(* IEC 61131-3 sources: Std_PalletMover/Class/MQTTClient_Interface (part 2) *)

      DiagnosticData.LogEvents.Level_Warning  := DiagnosticData.LogEvents.Level_Error;
      DiagnosticData.LogEvents.Level_Info     := DiagnosticData.LogEvents.Level_Error;
      DiagnosticData.LogEvents.Level_Debug    := DiagnosticData.LogEvents.Level_Error;

  end_if;

END_FUNCTION

FUNCTION MQTTClient_Interface::InitMem

END_FUNCTION
//================================================================================================================================================================
//----------------------------------------------------------------END OF INITITALISE METHODS----------------------------------------------------------------------
//================================================================================================================================================================

//================================================================================================================================================================
//-----------------------------------------------------------------SERVER INTERFACE METHODS-----------------------------------------------------------------------
//================================================================================================================================================================
FUNCTION VIRTUAL GLOBAL MQTTClient_Interface::ClientID::Read
	VAR_OUTPUT
		output (EAX) 	: UDINT;
	END_VAR

	ClientID := MQTTClient.ClientID.Read();
	output := ClientID;

END_FUNCTION

FUNCTION VIRTUAL GLOBAL MQTTClient_Interface::ClientID::Write
	VAR_INPUT
		input (EAX) 	: UDINT;
	END_VAR
	VAR_OUTPUT
		result (EAX) 	: UDINT;
	END_VAR

	ClientID := input;
	result := (MQTTClient.ClientID.Write(ClientID))$UDINT;

END_FUNCTION

FUNCTION VIRTUAL GLOBAL MQTTClient_Interface::XMLFilename::Read
	VAR_OUTPUT
		output (EAX) 	: UDINT;
	END_VAR

	XMLFilename := XMLFilenameString.Data.Read();
	output := XMLFilename;

END_FUNCTION

FUNCTION VIRTUAL GLOBAL MQTTClient_Interface::XMLFilename::Write
	VAR_INPUT
		input (EAX) 	: UDINT;
	END_VAR
	VAR_OUTPUT
		result (EAX) 	: UDINT;
	END_VAR

	XMLFilename := input;
	result := (XMLFilenameString.Data.Write(XMLFilename))$UDINT;

END_FUNCTION

FUNCTION VIRTUAL GLOBAL MQTTClient_Interface::ClientActive::Write
	VAR_INPUT
		input (EAX) 	: DINT;
	END_VAR
	VAR_OUTPUT
		result (EAX) 	: DINT;
	END_VAR
  VAR
  	iRetCode : INT;
    tmpPara : DINT;
  END_VAR

  //Falling edge (Disabling Client)
  if (ClientActive = 1) &
     (input = 0)        then

    //If the state is OK
    if InterfaceState = MCIS_Connected         |
       InterfaceState = MCIS_WaitForConnection |
       InterfaceState = MCIS_Reconnecting      then

      //Issue Disconnect Command
      iRetCode := MQTTClient.mqtt_disconnect();

      //Diagnostic Info:
      Diagnostic_Event( Event   :=  DL_LastErrorCode,
                        udValue :=  iRetCode$UDINT);

      if iRetCode <> MQTTClient::MQTT_ERR_SUCCESS$INT then
        Diagnostic_Event( Event   :=  DL_Error,
                          udValue :=  0);
      end_if;

      if iRetCode = MQTTClient::MQTT_ERR_SUCCESS$INT then
        //Create Log: MQTT Client disconnect requested

        Logging_InterfLog(usLevel     :=  MQTTCLIENTINTERFACE_LOGGING_LEVEL_DEBUG,
                          dMsgGroup   :=  MQCLIINF_LOG_DEBUG_CLIENTACTIVE_DISCONNECT_REQUESTED_GRP,
                          dMsgNbr     :=  MQCLIINF_LOG_DEBUG_CLIENTACTIVE_DISCONNECT_REQUESTED_MSG,
                          pMsg        :=  MQCLIINF_LOG_DEBUG_CLIENTACTIVE_DISCONNECT_REQUESTED_TEXT,
                          pPara1      :=  NIL,
                          pPara2      :=  NIL,
                          pPara3      :=  NIL,
                          pPara4      :=  NIL);

      elsif iRetCode = MQTTClient::MQTT_ERR_NO_CONN$INT then
        //Create Log: Requesting MQTT Client Disconnect Failed, no Connection to disconnect.

        Logging_InterfLog(usLevel     :=  MQTTCLIENTINTERFACE_LOGGING_LEVEL_WARNING,
                          dMsgGroup   :=  MQCLIINF_LOG_WARNING_CLIENTACTIVE_DISCONNECT_REQUESTED_GRP,
                          dMsgNbr     :=  MQCLIINF_LOG_WARNING_CLIENTACTIVE_DISCONNECT_REQUESTED_MSG,
                          pMsg        :=  MQCLIINF_LOG_WARNING_CLIENTACTIVE_DISCONNECT_REQUESTED_TEXT,
                          pPara1      :=  NIL,
                          pPara2      :=  NIL,
                          pPara3      :=  NIL,
                          pPara4      :=  NIL);

      else
        //Create Log: Unexpected retcode whilst requesting MQTT Client Disconnect.
        tmpPara := to_dint(iRetCode);

        Logging_InterfLog(usLevel     :=  MQTTCLIENTINTERFACE_LOGGING_LEVEL_ERR,
                          dMsgGroup   :=  MQCLIINF_LOG_WARNING_CLIENTACTIVE_DISCONNECT_UNEXPECTED_RETCODE_GRP,
                          dMsgNbr     :=  MQCLIINF_LOG_WARNING_CLIENTACTIVE_DISCONNECT_UNEXPECTED_RETCODE_MSG,
                          pMsg        :=  MQCLIINF_LOG_WARNING_CLIENTACTIVE_DISCONNECT_UNEXPECTED_RETCODE_TEXT,
                          pPara1      :=  #tmpPara,
                          pPara2      :=  NIL,
                          pPara3      :=  NIL,
                          pPara4      :=  NIL);
      end_if;

    end_if;

    ClientActive := 0;

  else

    ClientActive := input;

  end_if;

	result := ClientActive;

END_FUNCTION
//================================================================================================================================================================
//--------------------------------------------------------------END OF SERVER INTERFACE METHODS-------------------------------------------------------------------
//================================================================================================================================================================

//================================================================================================================================================================
//-----------------------------------------------------------------------CYCLIC METHODS---------------------------------------------------------------------------
//================================================================================================================================================================
FUNCTION VIRTUAL GLOBAL MQTTClient_Interface::CyWork
	VAR_INPUT
		EAX 	: UDINT;
	END_VAR
	VAR_OUTPUT
		state (EAX) 	: UDINT;
	END_VAR

	state := READY;
  MQTTClientInterfaceTask();

END_FUNCTION

FUNCTION MQTTClient_Interface::MQTTClientInterfaceTask
  VAR
  	iRetCode : INT;
    dTemp : DINT;
  END_VAR

  //Set FirstCall if state is changed
  Config.bFirstCall := InterfaceState <> LastState;

  //If not already in Error state, check for errors from interfaces
  if InterfaceState <> MCIS_Error then
    Diagnostic_ReadErrors();
  end_if;

  //=============================================
  //FSM For MQTT Client Interface
  //=============================================
  case InterfaceState of

    //-----------------------------------------------------------------
    //Wait for activation
    //-----------------------------------------------------------------
  	MQTTClient_Interface::t_e_MQTTClientStates::MCIS_Ready:

      if ClientActive = 1 then

        if Config.IsConn.PubTimeout then
          cDataMapPubTimeout := cDataMapPubTimeout.Read();
        end_if;

        if Config.IsConn.SubTimeout then
          cDataMapSubTimeout := cDataMapSubTimeout.Read();
        end_if;

        if Config.IsConn.ConnTimeout then
          cConnectTimeout := cConnectTimeout.Read();
        end_if;

        Logging_InterfLog(usLevel     :=  MQTTCLIENTINTERFACE_LOGGING_LEVEL_INFO,
                          dMsgGroup   :=  MQCLIINF_LOG_INFO_FSM_CLIENT_ACTIVATED_GRP,
                          dMsgNbr     :=  MQCLIINF_LOG_INFO_FSM_CLIENT_ACTIVATED_MSG,
                          pMsg        :=  MQCLIINF_LOG_INFO_FSM_CLIENT_ACTIVATED_TEXT,
                          pPara1      :=  NIL,
                          pPara2      :=  NIL,
                          pPara3      :=  NIL,
                          pPara4      :=  NIL);

        InterfaceState := MCIS_Initialise;

        //Reset Diagnostic Data
        Diagnostic_Event( Event   :=  DL_Reset,
                          udValue :=  0);
      end_if;

      LastState := MCIS_Ready;

    //-----------------------------------------------------------------
    //Initialise, Prepare, Read XML
    //-----------------------------------------------------------------
  	MQTTClient_Interface::t_e_MQTTClientStates::MCIS_Initialise:

      //Perform Init task
      case MCIT_Initialise(bFirstCall:=Config.bFirstCall) of

        TR_Busy:  //Stay in this state

        TR_Done:  //Next State

          InterfaceState := MCIS_Prepare;

        TR_Error: //Go to Error State

          InterfaceState := MCIS_Error;

      end_case;

      LastState := MCIS_Initialise;

    //-----------------------------------------------------------------
    //Prepare Connection, set parameters, initiate Connection
    //-----------------------------------------------------------------
  	MQTTClient_Interface::t_e_MQTTClientStates::MCIS_Prepare:

      //Perform Prepare task
      case MCIT_Prepare(bFirstCall:=Config.bFirstCall) of

        TR_Busy:  //Stay in this state

        TR_Done:  //Create Connection & Next State

          udTimestamp := ops.tAbsolute;

          MQTTClient.mqtt_loop_start();

          iRetCode := MQTTClient.mqtt_connect_async(  host      :=  #MQTTClientConfigData.Config.Connect.aHostname[0],
                                                      port      :=  MQTTClientConfigData.Config.Connect.iPort,
                                                      keepalive :=  MQTTClientConfigData.Config.Connect.iKeepalive);

          //Diagnostic Info:
          Diagnostic_Event( Event   :=  DL_LastErrorCode,
                            udValue :=  iRetCode$UDINT);

          if iRetCode = MQTTClient::MQTT_ERR_SUCCESS$INT then

            InterfaceState := MCIS_WaitForConnection;
            udTimestamp := ops.tAbsolute;

          else

            //Diagnostic Info:
            Diagnostic_Event( Event   :=  DL_Error,
                              udValue :=  0);

            Diagnostic_Event( Event   :=  DL_ConnectFail,
                              udValue :=  0);

            dTemp := to_dint(iRetCode);

            //Create Log Message
            Logging_InterfLog(usLevel     :=  MQTTCLIENTINTERFACE_LOGGING_LEVEL_ERR,
                              dMsgGroup   :=  MQCLIINF_LOG_ERROR_FSM_CONNECTION_FAILED_GRP,
                              dMsgNbr     :=  MQCLIINF_LOG_ERROR_FSM_CONNECTION_FAILED_MSG,
                              pMsg        :=  MQCLIINF_LOG_ERROR_FSM_CONNECTION_FAILED_TEXT,
                              pPara1      :=  #dTemp,
                              pPara2      :=  NIL,
                              pPara3      :=  NIL,
                              pPara4      :=  NIL);

            //Go to Error
            InterfaceState := MCIS_Error;

          end_if;

        TR_Error: //Go to Error State

          InterfaceState := MCIS_Error;

      end_case;

      LastState := MCIS_Prepare;

    //-----------------------------------------------------------------
    //Wait for connection to be made
    //-----------------------------------------------------------------
  	MQTTClient_Interface::t_e_MQTTClientStates::MCIS_WaitForConnection:

      if ops.tAbsolute - udTimestamp >= cConnectTimeout then
        InterfaceState := MCIS_Error;
        //Diagnostic Info:
        Diagnostic_Event( Event   :=  DL_WatchdogTimeout,
                          udValue :=  0);
      end_if;

      LastState := MCIS_WaitForConnection;

    //-----------------------------------------------------------------
    //Wait for connection to be made
    //-----------------------------------------------------------------
  	MQTTClient_Interface::t_e_MQTTClientStates::MCIS_Reconnecting:

      Diagnostic_Calculate();

    //-----------------------------------------------------------------
    //Connected state
    //-----------------------------------------------------------------
  	MQTTClient_Interface::t_e_MQTTClientStates::MCIS_Connected:

      Diagnostic_Calculate();
      DataMap_ProcessMap();

      LastState := MCIS_Connected;

    //-----------------------------------------------------------------
    //Error Occured
    //-----------------------------------------------------------------
  	MQTTClient_Interface::t_e_MQTTClientStates::MCIS_Error:

      //If this is the first cycle in this state
      if LastState <> InterfaceState then
        MQTTClient.mqtt_disconnect();
        udTimestamp := ops.tAbsolute;
      end_if;

      //If Reset
      if (Reset = 1)                                    |
         (cAutoResetTime <> 0                         &
          ops.tAbsolute - udTimestamp >= cAutoResetTime) then
        Reset := 0;
        InterfaceState := MCIS_Ready;
      end_if;

      LastState := MCIS_Error;

  end_case;

END_FUNCTION

FUNCTION MQTTClient_Interface::MCIT_Initialise
  VAR_INPUT
    bFirstCall : BOOL;
  END_VAR
	VAR_OUTPUT
		eRet 	: t_e_TaskRet;
	END_VAR

  //Assume Busy
  eRet := TR_Busy;

  //If first call, restart the FSM
  if bFirstCall then
    States.Initialise := MCSI_Initialize;
  end_if;

  //============================================
  //Initialise FSM
  //============================================
  case States.Initialise of

    //----------------------------------
    //Prepare mem, name and XML Reader
    //----------------------------------
    t_e_MCSInit::MCSI_Initialize:

      //Clear Mem
      SigCLib.MemSet( dst :=  #MQTTClientConfigData,
                      c   :=  0x00,
                      len :=  sizeof(MQTTClientConfigData));

      //If using the XML File, process it
      if Config.IsConn.UseXML then
        cUseXML := cUseXML.Read();
      end_if;

      if cUseXML = 1 then

        //XML Filename
        SigCLib.MemSet( dst :=  #Config.Initialize.aXMLFilename,
                        c   :=  0x00,
                        len :=  sizeof(Config.Initialize.aXMLFilename));
        XMLFilenameString.ReadDataOff(udOff :=  0,
                                      pData :=  #Config.Initialize.aXMLFilename[0],
                                      udMax :=  MQTTCLIENTINTERFACE_MAX_XMLNAME_LEN);
        //Reset Reader
        _XMLReader.Reset();
        _XMLReader.FreeReader();

        States.Initialise := MCSI_ReadXML;

      //If not using the XML File, skip reading & Processing
      else

        States.Initialise := MCSI_AppliConfig;

      end_if;

      //Get Logging Config from Client
      if Config.IsConn.LogConfig then
        cLogConfig := cLogConfig.Read();
      end_if;

    //----------------------------------
    //Read the XML
    //----------------------------------
    t_e_MCSInit::MCSI_ReadXML:

      //Start XML File Read
      if _XMLReader.ReadFile(FileName:=#Config.Initialize.aXMLFilename[0]) then
        States.Initialise := MCSI_WaitForReadXML;
        udTimestamp := ops.tAbsolute;
      else
        //Create Log: Failed to read XML File

        Logging_InterfLog(usLevel     :=  MQTTCLIENTINTERFACE_LOGGING_LEVEL_ERR,
                          dMsgGroup   :=  MQCLIINF_LOG_ERROR_FSM_INIT_READ_FILE_FAILED_GRP,
                          dMsgNbr     :=  MQCLIINF_LOG_ERROR_FSM_INIT_READ_FILE_FAILED_MSG,
                          pMsg        :=  MQCLIINF_LOG_ERROR_FSM_INIT_READ_FILE_FAILED_TEXT,
                          pPara1      :=  NIL,
                          pPara2      :=  NIL,
                          pPara3      :=  NIL,
                          pPara4      :=  NIL);

        States.Initialise := MCSI_Error;
      end_if;

    //----------------------------------
    //Wait for read to finish
    //----------------------------------
    t_e_MCSInit::MCSI_WaitForReadXML:

      //Read Complete
      if _XMLReader.GetXmlState() = _XMLReader::XML_READ_STATE::_STRUCT_CREATED then

        States.Initialise := MCSI_PrepDataMap;

      //Read Error
      elsif _XMLReader.GetXmlState() = _XMLReader::XML_READ_STATE::_ERROR then

        States.Initialise := MCSI_Error;

      //Timeout
      elsif ops.tAbsolute - udTimestamp >= MQTTCLIENTINTERFACE_XML_MAX_READ_TIME then

        States.Initialise := MCSI_Error;

      end_if;

    //----------------------------------
    //Prepare the DataMap - Remove all datamap entries that belong to the XML
    //----------------------------------
    t_e_MCSInit::MCSI_PrepDataMap:

      if Config.pDataMapConfig = NIL then
        //Create Log: Could not initialise, Datamap memory is not OK.

        Logging_InterfLog(usLevel     :=  MQTTCLIENTINTERFACE_LOGGING_LEVEL_ERR,
                          dMsgGroup   :=  MQCLIINF_LOG_ERROR_FSM_INIT_DATAMAP_PTR_GRP,
                          dMsgNbr     :=  MQCLIINF_LOG_ERROR_FSM_INIT_DATAMAP_PTR_MSG,
                          pMsg        :=  MQCLIINF_LOG_ERROR_FSM_INIT_DATAMAP_PTR_TEXT,
                          pPara1      :=  NIL,
                          pPara2      :=  NIL,
                          pPara3      :=  NIL,
                          pPara4      :=  NIL);

        eRet := TR_Error;
        return;
      end_if;

      DataMap_Clear();

      eRet := TR_Busy;
      States.Initialise := MCSI_ProcessXML;

    //----------------------------------
    //Process the XML
    //----------------------------------
    t_e_MCSInit::MCSI_ProcessXML:

      //Process XML
      if ProcessXML() then

        //Update Log Config
        cLogConfig := MQTTClientConfigData.Config.Logging.bdActiveLogs;
        if Config.IsConn.LogConfig then
          cLogConfig.Write(input:=cLogConfig);
        end_if;

        States.Initialise := MCSI_AppliConfig;
        Config.ConfigObject.State := CO_ClientID;

      //Failed
      else

        States.Initialise := MCSI_Error;

      end_if;

    //----------------------------------
    //Call the application config object
    //----------------------------------
    t_e_MCSInit::MCSI_AppliConfig:

      //If an object is logged in
      if Config.ConfigObject.pThis then

        //Process the user config
        case ConfigObject_Process() of
          //------------
          //Keep Calling
          //------------
          TR_Busy:

            eRet := TR_Busy;

          //------------
          //Done, Advance
          //------------
          TR_Done:

            eRet := TR_Done;

          //------------
          //Error Occurred
          //------------
          TR_Error:

            States.Initialise := MCSI_Error;

        end_case;

      else

        eRet := TR_Done;

      end_if;

    //----------------------------------
    //Error Occurred
    //----------------------------------
    t_e_MCSInit::MCSI_Error:

      eRet := TR_Error;

  end_case;

END_FUNCTION

FUNCTION MQTTClient_Interface::MCIT_Prepare
	VAR_INPUT
		bFirstCall 	: BOOL;
	END_VAR
	VAR_OUTPUT
		eRet 	: t_e_TaskRet;
	END_VAR
  VAR
  	iRetCode              : INT;
    pCA, pCert, pKey, pPW : ^CHAR;
    tmpPayLoadSize        : UDINT;
    tmpPara1              : DINT;
    tmpPara2              : DINT;
    tmpPara3              : DINT;
    pID                   : ^UINT;
  END_VAR

  //Assume OK
  eRet := TR_Done;

  //==================================
  //Set the MQTT Class Parameters
  //==================================

    //---------------------------------
    //Client ID
    //---------------------------------
    if MQTTClientConfigData.Config.bClientIDSet then
      pID := #MQTTClientConfigData.Config.aClientID[0];
    else
      pID := NIL;
    end_if;

    iRetCode := MQTTClient.mqtt_reinitialise( id            :=  pID,
                                              clean_session :=  (CleanSession.Read() = 1));

    //Diagnostic Info:
    Diagnostic_Event( Event   :=  DL_LastErrorCode,
                      udValue :=  iRetCode$UDINT);

    if iRetCode <> MQTTClient::MQTT_ERR_SUCCESS$INT then
      Diagnostic_Event( Event   :=  DL_Error,
                        udValue :=  0);
    end_if;
    //- - - - - - - - - - - - - - - - - - - - -
    //Process Reponse
    //- - - - - - - - - - - - - - - - - - - - -
    case iRetCode$MQTTClient::t_e_MQTTErrors of
      //-  -  -  -  -  -  -  -  -  -
      //OK
      //-  -  -  -  -  -  -  -  -  -
      MQTTClient::MQTT_ERR_SUCCESS:

      //-  -  -  -  -  -  -  -  -  -
      //Not OK
      //-  -  -  -  -  -  -  -  -  -
      MQTTClient::MQTT_ERR_NOMEM:

        eRet := TR_Error;
        //Create Log: Error during setting MQTTClient Parameters from XML File, Setting ClientID Failed, Not Enough memory

        Logging_InterfLog(usLevel     :=  MQTTCLIENTINTERFACE_LOGGING_LEVEL_ERR,
                          dMsgGroup   :=  MQCLIINF_LOG_ERROR_FSM_PREP_INIT_FAIL_NOMEM_GRP,
                          dMsgNbr     :=  MQCLIINF_LOG_ERROR_FSM_PREP_INIT_FAIL_NOMEM_MSG,
                          pMsg        :=  MQCLIINF_LOG_ERROR_FSM_PREP_INIT_FAIL_NOMEM_TEXT,
                          pPara1      :=  NIL,
                          pPara2      :=  NIL,
                          pPara3      :=  NIL,
                          pPara4      :=  NIL);
        return;

      //-  -  -  -  -  -  -  -  -  -
      //
      //-  -  -  -  -  -  -  -  -  -
      MQTTClient::MQTT_ERR_INVAL:

        eRet := TR_Error;
        //Create Log: Error during setting MQTTClient Parameters from XML File, Setting ClientID Failed, Input Value / Client State Not OK

        Logging_InterfLog(usLevel     :=  MQTTCLIENTINTERFACE_LOGGING_LEVEL_ERR,
                          dMsgGroup   :=  MQCLIINF_LOG_ERROR_FSM_PREP_INIT_FAIL_INPUT_GRP,
                          dMsgNbr     :=  MQCLIINF_LOG_ERROR_FSM_PREP_INIT_FAIL_INPUT_MSG,
                          pMsg        :=  MQCLIINF_LOG_ERROR_FSM_PREP_INIT_FAIL_INPUT_TEXT,
                          pPara1      :=  NIL,
                          pPara2      :=  NIL,
                          pPara3      :=  NIL,
                          pPara4      :=  NIL);
        return;

    end_case;

    //---------------------------------
    //Connect -> Username & Password
    //---------------------------------
    if MQTTClientConfigData.Config.Connect.ValuesSet.Username then //&
       //MQTTClientConfigData.Config.Connect.ValuesSet.Password then

      iRetCode := MQTTClient.mqtt_username_pw_set(username    :=  #MQTTClientConfigData.Config.Connect.aUsername[0],
                                                  password    :=  #MQTTClientConfigData.Config.Connect.aPassword[0]$BYTE,
                                                  udPassLen   :=  (SigCLib.StrLen16(str0:=#MQTTClientConfigData.Config.Connect.aPassword[0])*sizeof(UINT)));

      //Diagnostic Info:
      Diagnostic_Event( Event   :=  DL_LastErrorCode,
                        udValue :=  iRetCode$UDINT);

      if iRetCode <> MQTTClient::MQTT_ERR_SUCCESS$INT then
        Diagnostic_Event( Event   :=  DL_Error,
                          udValue :=  0);
      end_if;

      //- - - - - - - - - - - - - - - - - - - - -
      //Process Reponse
      //- - - - - - - - - - - - - - - - - - - - -
      case iRetCode$MQTTClient::t_e_MQTTErrors of
        //-  -  -  -  -  -  -  -  -  -
        //OK
        //-  -  -  -  -  -  -  -  -  -
        MQTTClient::MQTT_ERR_SUCCESS:

        //-  -  -  -  -  -  -  -  -  -
        //Not OK
        //-  -  -  -  -  -  -  -  -  -
        MQTTClient::MQTT_ERR_NOMEM:

          eRet := TR_Error;
          //Create Log: Error during setting MQTTClient Parameters from XML File, Setting Username & Password Failed, Not Enough memory

          Logging_InterfLog(usLevel     :=  MQTTCLIENTINTERFACE_LOGGING_LEVEL_ERR,
                            dMsgGroup   :=  MQCLIINF_LOG_ERROR_FSM_PREP_USNPW_FAIL_NOMEM_GRP,
                            dMsgNbr     :=  MQCLIINF_LOG_ERROR_FSM_PREP_USNPW_FAIL_NOMEM_MSG,
                            pMsg        :=  MQCLIINF_LOG_ERROR_FSM_PREP_USNPW_FAIL_NOMEM_TEXT,
                            pPara1      :=  NIL,
                            pPara2      :=  NIL,
                            pPara3      :=  NIL,
                            pPara4      :=  NIL);
          return;

        //-  -  -  -  -  -  -  -  -  -
        //Not OK
        //-  -  -  -  -  -  -  -  -  -
        MQTTClient::MQTT_ERR_INVAL:

          eRet := TR_Error;
          //Create Log: Error during setting MQTTClient Parameters from XML File, Setting Username & Password Failed, Input Value / Client State Not OK

          Logging_InterfLog(usLevel     :=  MQTTCLIENTINTERFACE_LOGGING_LEVEL_ERR,
                            dMsgGroup   :=  MQCLIINF_LOG_ERROR_FSM_PREP_USNPW_FAIL_INPUT_GRP,
                            dMsgNbr     :=  MQCLIINF_LOG_ERROR_FSM_PREP_USNPW_FAIL_INPUT_MSG,
                            pMsg        :=  MQCLIINF_LOG_ERROR_FSM_PREP_USNPW_FAIL_INPUT_TEXT,
                            pPara1      :=  NIL,
                            pPara2      :=  NIL,
                            pPara3      :=  NIL,
                            pPara4      :=  NIL);
          return;

      end_case;

    end_if;

    //---------------------------------
    //Connect -> Max Inflight Messages
    //---------------------------------
    if MQTTClientConfigData.Config.Connect.ValuesSet.MaxInflight then

      iRetCode := MQTTClient.mqtt_max_inflight_messages_set(max_inflight_messages:=MQTTClientConfigData.Config.Connect.iMaxInflightMessages);

      //Diagnostic Info:
      Diagnostic_Event( Event   :=  DL_LastErrorCode,
                        udValue :=  iRetCode$UDINT);

      if iRetCode <> MQTTClient::MQTT_ERR_SUCCESS$INT then
        Diagnostic_Event( Event   :=  DL_Error,
                          udValue :=  0);
      end_if;

      //- - - - - - - - - - - - - - - - - - - - -
      //Process Reponse
      //- - - - - - - - - - - - - - - - - - - - -
      case iRetCode$MQTTClient::t_e_MQTTErrors of
        //-  -  -  -  -  -  -  -  -  -
        //OK
        //-  -  -  -  -  -  -  -  -  -
        MQTTClient::MQTT_ERR_SUCCESS:

        //-  -  -  -  -  -  -  -  -  -
        //Not OK
        //-  -  -  -  -  -  -  -  -  -
        MQTTClient::MQTT_ERR_INVAL:

          eRet := TR_Error;
          //Create Log: Error during setting MQTTClient Parameters from XML File, Setting Max Inflight Messages Failed, Input Value / Client State Not OK
          tmpPara1 := to_dint(MQTTClientConfigData.Config.Connect.iMaxInflightMessages);

          Logging_InterfLog(usLevel     :=  MQTTCLIENTINTERFACE_LOGGING_LEVEL_ERR,
                            dMsgGroup   :=  MQCLIINF_LOG_ERROR_FSM_PREP_SET_INFLIGHT_GRP,
                            dMsgNbr     :=  MQCLIINF_LOG_ERROR_FSM_PREP_SET_INFLIGHT_MSG,
                            pMsg        :=  MQCLIINF_LOG_ERROR_FSM_PREP_SET_INFLIGHT_TEXT,
                            pPara1      :=  #tmpPara1,
                            pPara2      :=  NIL,
                            pPara3      :=  NIL,
                            pPara4      :=  NIL);
          return;

      end_case;

    end_if;

    //---------------------------------
    //Will
    //---------------------------------
    if MQTTClientConfigData.Config.Will.ValuesSet.Topic       &
       MQTTClientConfigData.Config.Will.ValuesSet.Payload     &
       MQTTClientConfigData.Config.Will.ValuesSet.QoS         &
       MQTTClientConfigData.Config.Will.ValuesSet.RetainWill  then

      MQTTClient.mqtt_will_clear();

      tmpPayLoadSize := SigCLib.StrLen(str:=#MQTTClientConfigData.Config.Will.aPayload[0]);

      iRetCode := MQTTClient.mqtt_will_set( topic       :=  #MQTTClientConfigData.Config.Will.aTopic[0],
                                            payloadLen  :=  tmpPayLoadSize,
                                            payload     :=  #MQTTClientConfigData.Config.Will.aPayload[0]$BYTE,
                                            qos         :=  MQTTClientConfigData.Config.Will.iQoS,
                                            retain_will :=  MQTTClientConfigData.Config.Will.bRetain);

      //Diagnostic Info:
      Diagnostic_Event( Event   :=  DL_LastErrorCode,
                        udValue :=  iRetCode$UDINT);

      if iRetCode <> MQTTClient::MQTT_ERR_SUCCESS$INT then
        Diagnostic_Event( Event   :=  DL_Error,
                          udValue :=  0);
      end_if;

      //- - - - - - - - - - - - - - - - - - - - -
      //Process Reponse
      //- - - - - - - - - - - - - - - - - - - - -
      case iRetCode$MQTTClient::t_e_MQTTErrors of
        //-  -  -  -  -  -  -  -  -  -
        //OK
        //-  -  -  -  -  -  -  -  -  -
        MQTTClient::MQTT_ERR_SUCCESS:

        //-  -  -  -  -  -  -  -  -  -
        //Not OK
        //-  -  -  -  -  -  -  -  -  -
        MQTTClient::MQTT_ERR_NOMEM:

          eRet := TR_Error;
          //Create Log: Error during setting MQTTClient Parameters from XML File, Setting Will Failed, Not Enough memory

          Logging_InterfLog(usLevel     :=  MQTTCLIENTINTERFACE_LOGGING_LEVEL_ERR,
                            dMsgGroup   :=  MQCLIINF_LOG_ERROR_FSM_PREP_SET_WILL_NOMEM_GRP,
                            dMsgNbr     :=  MQCLIINF_LOG_ERROR_FSM_PREP_SET_WILL_NOMEM_MSG,
                            pMsg        :=  MQCLIINF_LOG_ERROR_FSM_PREP_SET_WILL_NOMEM_TEXT,
                            pPara1      :=  NIL,
                            pPara2      :=  NIL,
                            pPara3      :=  NIL,
                            pPara4      :=  NIL);
          return;

        //-  -  -  -  -  -  -  -  -  -
        //Not OK
        //-  -  -  -  -  -  -  -  -  -
        MQTTClient::MQTT_ERR_INVAL:

          eRet := TR_Error;
          //Create Log: Error during setting MQTTClient Parameters from XML File, Setting Will Failed, Input Value / Client State Not OK

          Logging_InterfLog(usLevel     :=  MQTTCLIENTINTERFACE_LOGGING_LEVEL_ERR,
                            dMsgGroup   :=  MQCLIINF_LOG_ERROR_FSM_PREP_SET_WILL_INPUT_GRP,
                            dMsgNbr     :=  MQCLIINF_LOG_ERROR_FSM_PREP_SET_WILL_INPUT_MSG,
                            pMsg        :=  MQCLIINF_LOG_ERROR_FSM_PREP_SET_WILL_INPUT_TEXT,
                            pPara1      :=  NIL,
                            pPara2      :=  NIL,
                            pPara3      :=  NIL,
                            pPara4      :=  NIL);
          return;

        //-  -  -  -  -  -  -  -  -  -
        //Not OK
        //-  -  -  -  -  -  -  -  -  -
        MQTTClient::MQTT_ERR_PAYLOAD_SIZE:

          eRet := TR_Error;
          //Create Log: Error during setting MQTTClient Parameters from XML File, Setting Will Failed, Invalid Payload Size

          Logging_InterfLog(usLevel     :=  MQTTCLIENTINTERFACE_LOGGING_LEVEL_ERR,
                            dMsgGroup   :=  MQCLIINF_LOG_ERROR_FSM_PREP_SET_WILL_PAYLOAD_GRP,
                            dMsgNbr     :=  MQCLIINF_LOG_ERROR_FSM_PREP_SET_WILL_PAYLOAD_MSG,
                            pMsg        :=  MQCLIINF_LOG_ERROR_FSM_PREP_SET_WILL_PAYLOAD_TEXT,
                            pPara1      :=  #tmpPayLoadSize$DINT,
                            pPara2      :=  NIL,
                            pPara3      :=  NIL,
                            pPara4      :=  NIL);

          return;

        //-  -  -  -  -  -  -  -  -  -
        //Not OK
        //-  -  -  -  -  -  -  -  -  -
        MQTTClient::MQTT_ERR_MALFORMED_UTF8:

          eRet := TR_Error;
          //Create Log: Error during setting MQTTClient Parameters from XML File, Setting Will Failed, Malformed UTF8

          Logging_InterfLog(usLevel     :=  MQTTCLIENTINTERFACE_LOGGING_LEVEL_ERR,
                            dMsgGroup   :=  MQCLIINF_LOG_ERROR_FSM_PREP_SET_WILL_UTF8_GRP,
                            dMsgNbr     :=  MQCLIINF_LOG_ERROR_FSM_PREP_SET_WILL_UTF8_MSG,
                            pMsg        :=  MQCLIINF_LOG_ERROR_FSM_PREP_SET_WILL_UTF8_TEXT,
                            pPara1      :=  NIL,
                            pPara2      :=  NIL,
                            pPara3      :=  NIL,
                            pPara4      :=  NIL);
          return;

      end_case;

    end_if;

    //---------------------------------
    //Reconnect
    //---------------------------------
    if MQTTClientConfigData.Config.Reconnect.ValuesSet.MinInterval      &
       MQTTClientConfigData.Config.Reconnect.ValuesSet.MaxInterval      &
       MQTTClientConfigData.Config.Reconnect.ValuesSet.ExponentialScale then

      iRetCode := MQTTClient.mqtt_reconnect_delay_set(reconnect_delay             :=  to_uint(MQTTClientConfigData.Config.Reconnect.iMinInterval),
                                                      reconnect_delay_max         :=  to_uint(MQTTClientConfigData.Config.Reconnect.iMaxInterval),
                                                      reconnect_exponential_delay :=  MQTTClientConfigData.Config.Reconnect.bExponential);
      //Diagnostic Info:
      Diagnostic_Event( Event   :=  DL_LastErrorCode,
                        udValue :=  iRetCode$UDINT);

      if iRetCode <> MQTTClient::MQTT_ERR_SUCCESS$INT then
        Diagnostic_Event( Event   :=  DL_Error,
                          udValue :=  0);
      end_if;

      //- - - - - - - - - - - - - - - - - - - - -
      //Process Reponse
      //- - - - - - - - - - - - - - - - - - - - -
      case iRetCode$MQTTClient::t_e_MQTTErrors of
        //-  -  -  -  -  -  -  -  -  -
        //OK
        //-  -  -  -  -  -  -  -  -  -
        MQTTClient::MQTT_ERR_SUCCESS:

        //-  -  -  -  -  -  -  -  -  -
        //Not OK
        //-  -  -  -  -  -  -  -  -  -
        MQTTClient::MQTT_ERR_INVAL:

          eRet := TR_Error;
          //Create Log: Error during setting MQTTClient Parameters from XML File, Setting Reconnect Parameters Failed, Input Value / Client State Not OK

          tmpPara1 := to_dint(MQTTClientConfigData.Config.Reconnect.iMinInterval);
          tmpPara2 := to_dint(MQTTClientConfigData.Config.Reconnect.iMaxInterval);
          tmpPara3 := to_dint(MQTTClientConfigData.Config.Reconnect.bExponential);

          Logging_InterfLog(usLevel     :=  MQTTCLIENTINTERFACE_LOGGING_LEVEL_ERR,
                            dMsgGroup   :=  MQCLIINF_LOG_ERROR_FSM_PREP_SET_RECONNECT_INPUT_GRP,
                            dMsgNbr     :=  MQCLIINF_LOG_ERROR_FSM_PREP_SET_RECONNECT_INPUT_MSG,
                            pMsg        :=  MQCLIINF_LOG_ERROR_FSM_PREP_SET_RECONNECT_INPUT_TEXT,
                            pPara1      :=  #tmpPara1,
                            pPara2      :=  #tmpPara2,
                            pPara3      :=  #tmpPara3,
                            pPara4      :=  NIL);

          return;

      end_case;

    end_if;

    //---------------------------------
    //TLS
    //---------------------------------

    if MQTTClientConfigData.Config.TLS.ValuesSet.TLS then

      pCA := pCert := pKey := pPW := NIL;

      if MQTTClientConfigData.Config.TLS.ValuesSet.CAFile then
        pCA := #MQTTClientConfigData.Config.TLS.aCAFile[0];
      end_if;
      if MQTTClientConfigData.Config.TLS.ValuesSet.CertFile then
        pCert := #MQTTClientConfigData.Config.TLS.aCertFile[0];
      end_if;
      if MQTTClientConfigData.Config.TLS.ValuesSet.KeyFile then
        pKey := #MQTTClientConfigData.Config.TLS.aKeyFile[0];
      end_if;
      if MQTTClientConfigData.Config.TLS.ValuesSet.Password then
        pPW := #MQTTClientConfigData.Config.TLS.aPassword[0];
      end_if;

      iRetCode := MQTTClient.mqtt_tls_set(cafile    :=  pCA,
                                          certfile  :=  pCert,
                                          keyfile   :=  pKey,
                                          pw        :=  pPW);

      //Diagnostic Info:
      Diagnostic_Event( Event   :=  DL_LastErrorCode,
                        udValue :=  iRetCode$UDINT);

      if iRetCode <> MQTTClient::MQTT_ERR_SUCCESS$INT then
        Diagnostic_Event( Event   :=  DL_Error,
                          udValue :=  0);
      end_if;

      //- - - - - - - - - - - - - - - - - - - - -
      //Process Reponse
      //- - - - - - - - - - - - - - - - - - - - -
      case iRetCode$MQTTClient::t_e_MQTTErrors of
        //-  -  -  -  -  -  -  -  -  -
        //OK
        //-  -  -  -  -  -  -  -  -  -
        MQTTClient::MQTT_ERR_SUCCESS:

        //-  -  -  -  -  -  -  -  -  -
        //Not OK
        //-  -  -  -  -  -  -  -  -  -
        MQTTClient::MQTT_ERR_NOMEM:

          eRet := TR_Error;
          //Create Log: Error during setting MQTTClient Parameters from XML File, Setting TLS Data Failed, Not Enough memory

          Logging_InterfLog(usLevel     :=  MQTTCLIENTINTERFACE_LOGGING_LEVEL_ERR,
                            dMsgGroup   :=  MQCLIINF_LOG_ERROR_FSM_PREP_SET_TLS_NOMEM_GRP,
                            dMsgNbr     :=  MQCLIINF_LOG_ERROR_FSM_PREP_SET_TLS_NOMEM_MSG,
                            pMsg        :=  MQCLIINF_LOG_ERROR_FSM_PREP_SET_TLS_NOMEM_TEXT,
                            pPara1      :=  NIL,
                            pPara2      :=  NIL,
                            pPara3      :=  NIL,
                            pPara4      :=  NIL);
          return;

        //-  -  -  -  -  -  -  -  -  -
        //Not OK
        //-  -  -  -  -  -  -  -  -  -
        MQTTClient::MQTT_ERR_INVAL:

          eRet := TR_Error;
          //Create Log: Error during setting MQTTClient Parameters from XML File, Setting TLS Data Failed, Input Value / Client State Not OK

          Logging_InterfLog(usLevel     :=  MQTTCLIENTINTERFACE_LOGGING_LEVEL_ERR,
                            dMsgGroup   :=  MQCLIINF_LOG_ERROR_FSM_PREP_SET_TLS_INPUT_GRP,
                            dMsgNbr     :=  MQCLIINF_LOG_ERROR_FSM_PREP_SET_TLS_INPUT_MSG,
                            pMsg        :=  MQCLIINF_LOG_ERROR_FSM_PREP_SET_TLS_INPUT_TEXT,
                            pPara1      :=  NIL,
                            pPara2      :=  NIL,
                            pPara3      :=  NIL,
                            pPara4      :=  NIL);
          return;

      end_case;

    end_if;

    //===================
    //Set Callbacks
    //===================
    MQTTClient.mqtt_connect_with_flags_callback_set(  pThis                 :=  this,
                                                      on_connect_with_flags :=  #Callback_OnConnectWithFlags());
    MQTTClient.mqtt_disconnect_callback_set(          pThis                 :=  this,
                                                      on_disconnect         :=  #Callback_OnDisconnect());
    MQTTClient.mqtt_publish_callback_set(             pThis                 :=  this,
                                                      on_publish            :=  #Callback_OnPublish());
    MQTTClient.mqtt_message_callback_set(             pThis                 :=  this,
                                                      on_message            :=  #Callback_OnMessage());
    MQTTClient.mqtt_subscribe_callback_set(           pThis                 :=  this,
                                                      on_subscribe          :=  #Callback_OnSubscribe());
    MQTTClient.mqtt_unsubscribe_callback_set(         pThis                 :=  this,
                                                      on_unsubscribe        :=  #Callback_OnUnsubscribe());
    MQTTClient.mqtt_log_callback_set(                 pThis                 :=  this,
                                                      on_log                :=  #Callback_OnLog());
    MQTTClient.mqtt_log_with_detail_callback_set(     pThis                 :=  this,
                                                      on_log_with_detail    :=  #Callback_OnLog_WithDetail());

    //===================
    //Set Logging Filter
    //===================
    if MQTTClientConfigData.Config.Logging.bLogSet then
      _ComLogging.FileLogLevel.Write(input:=MQTTClientConfigData.Config.Logging.bdActiveLogs$UDINT);
      _ComLogging.EventLogLevel.Write(input:=MQTTClientConfigData.Config.Logging.bdActiveLogs$UDINT);
    end_if;

END_FUNCTION
//================================================================================================================================================================
//-------------------------------------------------------------------END OF CYCLIC METHODS------------------------------------------------------------------------
//================================================================================================================================================================

//================================================================================================================================================================
//---------------------------------------------------------------------INTERFACE METHODS--------------------------------------------------------------------------
//================================================================================================================================================================
FUNCTION GLOBAL MQTTClient_Interface::MQTT_Subscribe
	VAR_INPUT
		pTopic 	: ^UINT;
		iQoS 	: INT;
		pThis 	: ^void;
		pCallback 	: ^void;
		pMid 	: ^INT;
		pApplMsgID 	: ^UDINT;
	END_VAR
	VAR_OUTPUT
		retCode 	: INT;
	END_VAR
  VAR
  	iThisMID : INT;
    udThisApplID : UDINT;
    tmpPara, tmpPara2 : DINT;
    pEntry : ^t_s_PubSubEntry;
  END_VAR

  //Assume Error
  retCode := MQTT_ERR_INVAL;

  CriticalSection.SectionStart();

  //Diagnostic Info
  Diagnostic_Event( Event   :=  DL_SubRequest,
                    udValue :=  0);

  //If the input values are not OK
  if pTopic = NIL               |
     iQoS < MQTT_PROT_QOS_MIN   |
     iQoS > MQTT_PROT_QOS_MAX   |
     pThis = NIL                |
     pMid = NIL                 then
    //Create Log: Could not Issue Subscirbe Request, invalid input values.

    tmpPara := to_dint(iQoS);

    Logging_InterfLog(usLevel     :=  MQTTCLIENTINTERFACE_LOGGING_LEVEL_ERR,
                      dMsgGroup   :=  MQCLIINF_LOG_ERROR_SUBSCRIBE_SUB_FAILED_INVALID_INPUT_GRP,
                      dMsgNbr     :=  MQCLIINF_LOG_ERROR_SUBSCRIBE_SUB_FAILED_INVALID_INPUT_MSG,
                      pMsg        :=  MQCLIINF_LOG_ERROR_SUBSCRIBE_SUB_FAILED_INVALID_INPUT_TEXT,
                      pPara1      :=  #pTopic$DINT,
                      pPara2      :=  #tmpPara,
                      pPara3      :=  #pThis$DINT,
                      pPara4      :=  #pCallback$DINT);

    Diagnostic_Event( Event   :=  DL_SubFail,
                      udValue :=  0);

    CriticalSection.SectionStop();
    return;

  end_if;

  //If the interface is not in the correct state
  if InterfaceState < MCIS_Reconnecting |
     InterfaceState > MCIS_Connected    |
     Config.pPubSubConfig = NIL         then

    //Create Log: Could not issue Subscribe Request, The MQTT Interface is not initialized.

    Logging_InterfLog(usLevel     :=  MQTTCLIENTINTERFACE_LOGGING_LEVEL_ERR,
                      dMsgGroup   :=  MQCLIINF_LOG_ERROR_SUBSCRIBE_SUB_FAILED_INTERFACE_STATE_GRP,
                      dMsgNbr     :=  MQCLIINF_LOG_ERROR_SUBSCRIBE_SUB_FAILED_INTERFACE_STATE_MSG,
                      pMsg        :=  MQCLIINF_LOG_ERROR_SUBSCRIBE_SUB_FAILED_INTERFACE_STATE_TEXT,
                      pPara1      :=  #InterfaceState$DINT,
                      pPara2      :=  NIL,
                      pPara3      :=  NIL,
                      pPara4      :=  NIL);

    Diagnostic_Event( Event   :=  DL_SubFail,
                      udValue :=  0);

    CriticalSection.SectionStop();
    return;

  end_if;

  //If there is no more space in the list
  if Config.pPubSubConfig^.PubSubList.udNumEntries >= Config.pPubSubConfig^.PubSubList.udMaxEntries - 1 then

    retCode := MQTT_ERR_NOMEM;
    //Create Log: Could not issue subscribe request, MQTT Interface PubSubList is Full.

    tmpPara   := to_dint(Config.pPubSubConfig^.PubSubList.udMaxEntries);
    tmpPara2  := to_dint(Config.pPubSubConfig^.PubSubList.udNumEntries);

    Logging_InterfLog(usLevel     :=  MQTTCLIENTINTERFACE_LOGGING_LEVEL_ERR,
                      dMsgGroup   :=  MQCLIINF_LOG_ERROR_SUBSCRIBE_SUB_FAILED_LIST_FULL_GRP,
                      dMsgNbr     :=  MQCLIINF_LOG_ERROR_SUBSCRIBE_SUB_FAILED_LIST_FULL_MSG,
                      pMsg        :=  MQCLIINF_LOG_ERROR_SUBSCRIBE_SUB_FAILED_LIST_FULL_TEXT,
                      pPara1      :=  #tmpPara2,
                      pPara2      :=  #tmpPara,
                      pPara3      :=  NIL,
                      pPara4      :=  NIL);

    Diagnostic_Event( Event   :=  DL_SubFail,
                      udValue :=  0);

    CriticalSection.SectionStop();
    return;

  end_if;

  //========================
  //Add the QoS Diag Event
  //========================
  case iQos of
    //---------
    //QoS 0
    //---------
    0:
        Diagnostic_Event( Event   :=  DL_Sub0,
                          udValue :=  0);

    //---------
    //QoS 1
    //---------
    1:
        Diagnostic_Event( Event   :=  DL_Sub1,
                          udValue :=  0);

    //---------
    //QoS 2
    //---------
    2:
        Diagnostic_Event( Event   :=  DL_Sub2,
                          udValue :=  0);
  end_case;

  // Check if the subscription already exists, if so just return Already Subscribed
  udThisApplID := PubSub_CheckSubscription( pTopic    :=  pTopic,
                                            pThis     :=  pThis,
                                            pCallback :=  pCallback);

  if udThisApplID > 0 then

    tmpPara := to_dint(udThisApplID);

    Logging_InterfLog(usLevel     :=  MQTTCLIENTINTERFACE_LOGGING_LEVEL_INFO,
                      dMsgGroup   :=  MQCLIINF_LOG_INFO_SUBSCRIBE_ALREADY_SUBSCRIBED_GRP,
                      dMsgNbr     :=  MQCLIINF_LOG_INFO_SUBSCRIBE_ALREADY_SUBSCRIBED_MSG,
                      pMsg        :=  MQCLIINF_LOG_INFO_SUBSCRIBE_ALREADY_SUBSCRIBED_TEXT,
                      pPara1      :=  #tmpPara,
                      pPara2      :=  NIL,
                      pPara3      :=  NIL,
                      pPara4      :=  NIL);

    retCode := MQTTClient::MQTT_ERR_ALREADY_SUB;

    CriticalSection.SectionStop();
    return;

  end_if;

  iThisMID      := Counters_GetSubMID();
  udThisApplID  := Counters_GetApplID();

  //Subscribe
  retCode := MQTTClient.mqtt_subscribe(mid        :=  #iThisMID,
                                       subscribe  :=  pTopic,
                                       qos        :=  iQoS);

  //Diagnostic Info:
  Diagnostic_Event( Event   :=  DL_LastErrorCode,
                    udValue :=  retCode$UDINT);

  //If the MQTT Client accepts the subscription, log the subscription to the PubSub List
  if retCode = MQTT_ERR_SUCCESS$INT then

    pEntry := (Config.pPubSubConfig^.PubSubList.pEntries$UDINT + sizeof(t_s_PubSubEntry)*Config.pPubSubConfig^.PubSubList.udNumEntries)$^t_s_PubSubEntry;

    pEntry^.iMid             := iThisMID;
    pEntry^.EntryType        := PSE_Subscribe;
    pEntry^.Callback.pThis   := pThis;
    pEntry^.Callback.pMethod := pCallback;
    pEntry^.udAppliID        := udThisApplID;
    pEntry^.iUnsubMid        := -1;

    if pApplMsgID then
      pApplMsgID^ := udThisApplID;
    end_if;

    if pMid then
      pMid^ := iThisMID;
    end_if;

    SigCLib.MemSet( dst :=  #pEntry^.aTopic[0],
                    c   :=  0x00,
                    len :=  sizeof(t_s_PubSubEntry.aTopic));
    SigCLib.StrCpy16( dst0  :=  #pEntry^.aTopic[0],
                      src0  :=  pTopic);

    Config.pPubSubConfig^.PubSubList.udNumEntries += 1;
    Counters_IncSubMID();
    Counters_IncApplID();

    //Create Log: Successfully issued Subscribe Request.

    tmpPara := to_dint(iThisMID);

    Logging_InterfLog(usLevel     :=  MQTTCLIENTINTERFACE_LOGGING_LEVEL_INFO,
                      dMsgGroup   :=  MQCLIINF_LOG_INFO_SUBSCRIBE_ENTRY_ADDED_GRP,
                      dMsgNbr     :=  MQCLIINF_LOG_INFO_SUBSCRIBE_ENTRY_ADDED_MSG,
                      pMsg        :=  MQCLIINF_LOG_INFO_SUBSCRIBE_ENTRY_ADDED_TEXT,
                      pPara1      :=  #tmpPara,
                      pPara2      :=  NIL,
                      pPara3      :=  NIL,
                      pPara4      :=  NIL);

  else

    Logging_InterfLog(usLevel     :=  MQTTCLIENTINTERFACE_LOGGING_LEVEL_ERR,
                      dMsgGroup   :=  MQCLIINF_LOG_ERROR_SUBSCRIBE_SUB_FAILED_GRP,
                      dMsgNbr     :=  MQCLIINF_LOG_ERROR_SUBSCRIBE_SUB_FAILED_MSG,
                      pMsg        :=  MQCLIINF_LOG_ERROR_SUBSCRIBE_SUB_FAILED_TEXT,
                      pPara1      :=  #tmpPara,
                      pPara2      :=  NIL,
                      pPara3      :=  NIL,
                      pPara4      :=  NIL);

    //Diagnostic Data
    Diagnostic_Event( Event   :=  DL_Error,
                      udValue :=  0);
    Diagnostic_Event( Event   :=  DL_SubFail,
                      udValue :=  0);

  end_if;

  CriticalSection.SectionStop();

END_FUNCTION

FUNCTION GLOBAL MQTTClient_Interface::MQTT_Publish
	VAR_INPUT
		pTopic 	: ^UINT;
		iQoS 	: INT;
		pPayload 	: ^void;
		udPayloadLen 	: UDINT;
		bRetain 	: BOOL;
		pThis 	: ^void;
		pCallback 	: ^void;
		pMid 	: ^INT;
		pApplMsgID 	: ^UDINT;
	END_VAR
	VAR_OUTPUT
		retCode 	: INT;
	END_VAR
  VAR
    iRetCode : INT;
  	iThisMID : INT;
    udThisApplID : UDINT;
    tmpPara, tmpPara2 : DINT;
    pEntry : ^t_s_PubSubEntry;
  END_VAR

  CriticalSection.SectionStart();

  //Assume Fail
  retCode := MQTT_ERR_INVAL;

  Diagnostic_Event( Event   :=  DL_PubRequest,
                    udValue :=  0);

  //Check input values
  if pTopic = NIL                                                                 |
     SigCLib.StrLen16(str0:=pTopic) > MQTTCLIENTINTERFACE_PUBSUB_TOPIC_MAX_LEN    |
     iQoS > MQTT_PROT_QOS_MAX                                                     |
     iQos < MQTT_PROT_QOS_MIN                                                     |
     udPayloadLen > MQTTCLIENT_MAX_DATA_LEN                                       |
     ((pPayload <> NIL) & (udPayloadLen = 0))                                     then
    //Create Log: Failed to issue publish request, invalid input values.

    tmpPara := to_dint(iQoS);

    Logging_InterfLog(usLevel     :=  MQTTCLIENTINTERFACE_LOGGING_LEVEL_ERR,
                      dMsgGroup   :=  MQCLIINF_LOG_ERROR_PUBLISH_PUB_FAILED_INVALID_INPUT_GRP,
                      dMsgNbr     :=  MQCLIINF_LOG_ERROR_PUBLISH_PUB_FAILED_INVALID_INPUT_MSG,
                      pMsg        :=  MQCLIINF_LOG_ERROR_PUBLISH_PUB_FAILED_INVALID_INPUT_TEXT,
                      pPara1      :=  #pTopic$DINT,
                      pPara2      :=  #tmpPara,
                      pPara3      :=  #udPayloadLen$DINT,
                      pPara4      :=  #pPayload$DINT);

    Diagnostic_Event( Event   :=  DL_PubFail,
                      udValue :=  0);

    return;

  end_if;

  //Check the state
  if InterfaceState < MCIS_Reconnecting |
     InterfaceState > MCIS_Connected    |
     Config.pPubSubConfig = NIL         then

    retCode := MQTT_ERR_NO_CONN;

    //Create Log: Failed to issue publish request, no Connection MQTT Broker or the MQTT interface class is not initialised.

    Logging_InterfLog(usLevel     :=  MQTTCLIENTINTERFACE_LOGGING_LEVEL_ERR,
                      dMsgGroup   :=  MQCLIINF_LOG_ERROR_PUBLISH_PUB_FAILED_INTERFACE_STATE_GRP,
                      dMsgNbr     :=  MQCLIINF_LOG_ERROR_PUBLISH_PUB_FAILED_INTERFACE_STATE_MSG,
                      pMsg        :=  MQCLIINF_LOG_ERROR_PUBLISH_PUB_FAILED_INTERFACE_STATE_TEXT,
                      pPara1      :=  #InterfaceState$DINT,
                      pPara2      :=  NIL,
                      pPara3      :=  NIL,
                      pPara4      :=  NIL);

    Diagnostic_Event( Event   :=  DL_PubFail,
                      udValue :=  0);

    return;

  end_if;

  //If there is no more space in the list
  if Config.pPubSubConfig^.PubSubList.udNumEntries >= Config.pPubSubConfig^.PubSubList.udMaxEntries - 1 then

    retCode := MQTT_ERR_NOMEM;

    Diagnostic_Event( Event   :=  DL_PubFail,
                      udValue :=  0);

    tmpPara   := to_dint(Config.pPubSubConfig^.PubSubList.udMaxEntries);
    tmpPara2  := to_dint(Config.pPubSubConfig^.PubSubList.udNumEntries);

    Logging_InterfLog(usLevel     :=  MQTTCLIENTINTERFACE_LOGGING_LEVEL_ERR,
                      dMsgGroup   :=  MQCLIINF_LOG_ERROR_SUBSCRIBE_SUB_FAILED_LIST_FULL_GRP,
                      dMsgNbr     :=  MQCLIINF_LOG_ERROR_SUBSCRIBE_SUB_FAILED_LIST_FULL_MSG,
                      pMsg        :=  MQCLIINF_LOG_ERROR_SUBSCRIBE_SUB_FAILED_LIST_FULL_TEXT,
                      pPara1      :=  #tmpPara2,
                      pPara2      :=  #tmpPara,
                      pPara3      :=  NIL,
                      pPara4      :=  NIL);

    return;

  end_if;

  udThisApplID  := Counters_GetApplID();

  iRetCode := MQTTClient.mqtt_publish(mid         :=  #iThisMID,
                                      topic       :=  pTopic,
                                      payloadLen  :=  udPayloadLen,
                                      payload     :=  pPayload,
                                      qos         :=  iQoS,
                                      retain_pub  :=  bRetain);

  //Diagnostic Info:
  Diagnostic_Event( Event   :=  DL_LastErrorCode,
                    udValue :=  retCode$UDINT);

  if iRetCode <> MQTT_ERR_SUCCESS$INT then

    retCode := iRetCode;

    tmpPara := to_dint(retCode);

    Logging_InterfLog(usLevel     :=  MQTTCLIENTINTERFACE_LOGGING_LEVEL_ERR,
                      dMsgGroup   :=  MQCLIINF_LOG_ERROR_SUBSCRIBE_SUB_FAILED_GRP,
                      dMsgNbr     :=  MQCLIINF_LOG_ERROR_SUBSCRIBE_SUB_FAILED_MSG,
                      pMsg        :=  MQCLIINF_LOG_ERROR_SUBSCRIBE_SUB_FAILED_TEXT,
                      pPara1      :=  #tmpPara,
                      pPara2      :=  NIL,
                      pPara3      :=  NIL,
                      pPara4      :=  NIL);

    Diagnostic_Event( Event   :=  DL_PubFail,
                      udValue :=  0);

    Diagnostic_Event( Event   :=  DL_Error,
                      udValue :=  0);

    return;

  end_if;

  Counters_IncPubMID();
  Counters_IncApplID();

  //========================
  //Add the QoS Diag Event
  //========================
  case iQos of
    //---------
    //QoS 0
    //---------
    0:
        Diagnostic_Event( Event   :=  DL_Pub0,
                          udValue :=  0);

    //---------
    //QoS 1
    //---------
    1:
        Diagnostic_Event( Event   :=  DL_Pub1,
                          udValue :=  0);

    //---------
    //QoS 2
    //---------
    2:
        Diagnostic_Event( Event   :=  DL_Pub2,
                          udValue :=  0);
  end_case;

  Diagnostic_Event( Event   :=  DL_TXBytes,
                    udValue :=  udPayloadLen);

  //Add to the PubSubList

  pEntry := (Config.pPubSubConfig^.PubSubList.pEntries$UDINT + sizeof(t_s_PubSubEntry)*Config.pPubSubConfig^.PubSubList.udNumEntries)$^t_s_PubSubEntry;

  pEntry^.iMid             := iThisMID;
  pEntry^.EntryType        := PSE_Publish;
  pEntry^.udAppliID        := udThisApplID;
  pEntry^.Callback.pThis   := pThis;
  pEntry^.Callback.pMethod := pCallback;
  pEntry^.iUnsubMid        := -1;

  SigCLib.MemSet( dst :=  #pEntry^.aTopic,
                  c   :=  0x00,
                  len :=  sizeof(t_s_PubSubEntry.aTopic));

  SigCLib.StrCpy16( dst0  :=  #pEntry^.aTopic[0],
                    src0  :=  pTopic);

  if pMid then
    pMid^ := iThisMID;
  end_if;
  if pApplMsgID then
    pApplMsgID^:= udThisApplID;
  end_if;

  Config.pPubSubConfig^.PubSubList.udNumEntries += 1;

  retCode := MQTT_ERR_SUCCESS;

  CriticalSection.SectionStop();

END_FUNCTION

FUNCTION GLOBAL MQTTClient_Interface::MQTT_Unsubscribe
	VAR_INPUT
		pApplMsgID 	: ^UDINT;
		pTopic 	: ^UINT;
		pMid 	: ^INT;
		pThis 	: ^void;
		pCallback 	: ^void;
	END_VAR
	VAR_OUTPUT
		retCode 	: INT;
	END_VAR
  VAR
    iThisMID : INT;
  	udApplMsgID, udCount, udCount2 : UDINT;
    pPubSubEntry, pPubSubSearchEntry : ^t_s_PubSubEntry;
    bTopicFound, bSubscriptionFound : BOOL;
    tmpPara : DINT;
  END_VAR

  //Assume Error
  retCode := MQTT_ERR_INVAL;

  Diagnostic_Event( Event   :=  DL_UnsubRequest,
                    udValue :=  0);

  //If the input is oK
  if (pApplMsgID | pTopic)                                &
     Config.pPubSubConfig                                 &
     (Config.pPubSubConfig^.PubSubList.udNumEntries > 0)  then

    udApplMsgID := 0;
    bTopicFound := TRUE;

    //1. Determine the Application Message ID:

    //==========================================================
    //Based on the input, determine the ApplMsgID to Unsubscribe
    //==========================================================
      //-----------------------------------
      //Both are set, Use the ApplMsgID
      //-----------------------------------
      if pApplMsgID &
         pTopic then

        udApplMsgID := pApplMsgID^;

      //-----------------------------------
      //Only ApplMsgID is set, use this
      //-----------------------------------
      elsif pApplMsgID      &
            (pTopic = NIL)  then

        udApplMsgID := pApplMsgID^;

      //-----------------------------------
      //Only Topic is set, Determine ApplMsgID
      //-----------------------------------
      elsif pTopic              &
            (pApplMsgID = NIL)  then

        pPubSubEntry := Config.pPubSubConfig^.PubSubList.pEntries;

        for udCount := 0 to Config.pPubSubConfig^.PubSubList.udNumEntries - 1 do

          if SigCLib.StrCmp16(src1:=pTopic, src2:=#pPubSubEntry^.aTopic[0]) = 0 then
            udApplMsgID := pPubSubEntry^.udAppliID;
            bTopicFound := TRUE;
            exit;
          end_if;

          pPubSubEntry$UDINT += sizeof(t_s_PubSubEntry);

        end_for;

        if bTopicFound = FALSE then
          //Create Log: Failed to perform Unsubscribe command, Could not find the Subscription in the PubSubList.

          Logging_InterfLog(usLevel     :=  MQTTCLIENTINTERFACE_LOGGING_LEVEL_ERR,
                            dMsgGroup   :=  MQCLIINF_LOG_ERROR_UNSUBSCRIBE_UNSUB_FAILED_NOT_FOUND_GRP,
                            dMsgNbr     :=  MQCLIINF_LOG_ERROR_UNSUBSCRIBE_UNSUB_FAILED_NOT_FOUND_MSG,
                            pMsg        :=  MQCLIINF_LOG_ERROR_UNSUBSCRIBE_UNSUB_FAILED_NOT_FOUND_TEXT,
                            pPara1      :=  NIL,
                            pPara2      :=  NIL,
                            pPara3      :=  NIL,
                            pPara4      :=  NIL);

          Diagnostic_Event( Event   :=  DL_UnsubFail,
                            udValue :=  0);

          return;
        end_if;

      end_if;

    //2. Find and Unsubscribe the Message

    pPubSubEntry := Config.pPubSubConfig^.PubSubList.pEntries;

    for udCount := 0 to Config.pPubSubConfig^.PubSubList.udNumEntries - 1 do

      if pPubSubEntry^.udAppliID = udApplMsgID then

        //See if this topic is still subscribed to by any other parties, if so, do not unsubscribe
        bSubscriptionFound := FALSE;

        pPubSubSearchEntry$UDINT := (Config.pPubSubConfig^.PubSubList.pEntries)$UDINT;

        for udCount2 := 0 to Config.pPubSubConfig^.PubSubList.udNumEntries - 1 do

          if (udCount2 <> udCount) &
             SigCLib.StrCmp16(src1:=#pPubSubEntry^.aTopic[0], src2:=#pPubSubSearchEntry^.aTopic[0]) = 0 then

            //Create Log: Unsubscribe: Unsubscribe requested for a topic where atleast one other party in the application is still subscribed, the Unsubscribe request will not be sent
            Logging_InterfLog(usLevel     :=  MQTTCLIENTINTERFACE_LOGGING_LEVEL_DEBUG,
                              dMsgGroup   :=  MQCLIINF_LOG_DEBUG_UNSUBSCRIBE_STILL_SUBSCRIBED_GRP,
                              dMsgNbr     :=  MQCLIINF_LOG_DEBUG_UNSUBSCRIBE_STILL_SUBSCRIBED_MSG,
                              pMsg        :=  MQCLIINF_LOG_DEBUG_UNSUBSCRIBE_STILL_SUBSCRIBED_TEXT,
                              pPara1      :=  #pPubSubEntry^.udAppliID$DINT,
                              pPara2      :=  #pPubSubSearchEntry^.udAppliID$DINT,
                              pPara3      :=  NIL,
                              pPara4      :=  NIL);

            bSubscriptionFound := TRUE;
            exit;

          end_if;

          pPubSubSearchEntry$UDINT += sizeof(t_s_PubSubEntry);

        end_for;

        iThisMID := Counters_GetSubMID();

        pPubSubEntry^.iUnsubMid := iThisMID;

        if pMid then
          pMid^ := iThisMID;
        end_if;

        Counters_IncSubMID();

        //If no other subscription was found for this topic, unsubscribe
        if bSubscriptionFound = FALSE then

          retCode := MQTTClient.mqtt_unsubscribe( mid   :=  #pPubSubEntry^.iUnsubMid,
                                                  unsub :=  #pPubSubEntry^.aTopic[0]);

          //Diagnostic Info:
          Diagnostic_Event( Event   :=  DL_LastErrorCode,
                            udValue :=  retCode$UDINT);

          if retCode <> MQTTClient::MQTT_ERR_SUCCESS$INT then

            Diagnostic_Event( Event   :=  DL_UnsubFail,
                              udValue :=  0);
            Diagnostic_Event( Event   :=  DL_Error,
                              udValue :=  0);

          end_if;

          //====================
          //Act on RetCode
          //====================
          case retCode$MQTTClient::t_e_MQTTErrors of
            //-----------------
            //OK
            //-----------------
            MQTT_ERR_SUCCESS:

              //Save Callback Data if set
              if pCallback &
                 pThis     then

                pPubSubEntry^.Callback.pThis    := pThis;
                pPubSubEntry^.Callback.pMethod  := pCallback;

              //Callback data not set but also no pre-existing callback data, the user will receive no feedback
              elsif pPubSubEntry^.Callback.pThis    = NIL |
                    pPubSubEntry^.Callback.pMethod  = NIL then

                //Create Log: No Callback details specified during Unsubscribe, also no pre existing details, no callback possible.

                tmpPara := to_dint(iThisMID);

                Logging_InterfLog(usLevel     :=  MQTTCLIENTINTERFACE_LOGGING_LEVEL_WARNING,
                                  dMsgGroup   :=  MQCLIINF_LOG_WARNING_UNSUBSCRIBE_CALLBACK_NOTSET_GRP,
                                  dMsgNbr     :=  MQCLIINF_LOG_WARNING_UNSUBSCRIBE_CALLBACK_NOTSET_MSG,
                                  pMsg        :=  MQCLIINF_LOG_WARNING_UNSUBSCRIBE_CALLBACK_NOTSET_TEXT,
                                  pPara1      :=  #udApplMsgID$DINT,
                                  pPara2      :=  #tmpPara,
                                  pPara3      :=  NIL,
                                  pPara4      :=  NIL);

              end_if;

              //Create Log: Successfully issued the unsubscribe request for...

              tmpPara := to_dint(iThisMID);

              Logging_InterfLog(usLevel     :=  MQTTCLIENTINTERFACE_LOGGING_LEVEL_INFO,
                                dMsgGroup   :=  MQCLIINF_LOG_INFO_UNSUBSCRIBE_ENTRY_ADDED_GRP,
                                dMsgNbr     :=  MQCLIINF_LOG_INFO_UNSUBSCRIBE_ENTRY_ADDED_MSG,
                                pMsg        :=  MQCLIINF_LOG_INFO_UNSUBSCRIBE_ENTRY_ADDED_TEXT,
                                pPara1      :=  #udApplMsgID$DINT,
                                pPara2      :=  #tmpPara,
                                pPara3      :=  NIL,
                                pPara4      :=  NIL);

            //-----------------
            //Error
            //-----------------
            MQTT_ERR_INVAL:

              //Create Log: Unsubscribe failed, input values not accepted

              tmpPara := to_dint(iThisMID);

              Logging_InterfLog(usLevel     :=  MQTTCLIENTINTERFACE_LOGGING_LEVEL_ERR,
                                dMsgGroup   :=  MQCLIINF_LOG_ERROR_UNSUBSCRIBE_UNSUB_REQ_FAILED_INPUT_GRP,
                                dMsgNbr     :=  MQCLIINF_LOG_ERROR_UNSUBSCRIBE_UNSUB_REQ_FAILED_INPUT_MSG,
                                pMsg        :=  MQCLIINF_LOG_ERROR_UNSUBSCRIBE_UNSUB_REQ_FAILED_INPUT_TEXT,
                                pPara1      :=  #udApplMsgID$DINT,
                                pPara2      :=  #tmpPara,
                                pPara3      :=  NIL,
                                pPara4      :=  NIL);

            //-----------------
            //Retry
            //-----------------
            MQTT_ERR_NO_CONN:

              //Create Log: Unsubscribe failed, no connection mqtt client

              tmpPara := to_dint(iThisMID);

              Logging_InterfLog(usLevel     :=  MQTTCLIENTINTERFACE_LOGGING_LEVEL_ERR,
                                dMsgGroup   :=  MQCLIINF_LOG_ERROR_UNSUBSCRIBE_UNSUB_FAILED_CONN_GRP,
                                dMsgNbr     :=  MQCLIINF_LOG_ERROR_UNSUBSCRIBE_UNSUB_FAILED_CONN_MSG,
                                pMsg        :=  MQCLIINF_LOG_ERROR_UNSUBSCRIBE_UNSUB_FAILED_CONN_TEXT,
                                pPara1      :=  #udApplMsgID$DINT,
                                pPara2      :=  #tmpPara,
                                pPara3      :=  NIL,
                                pPara4      :=  NIL);

            //-----------------
            //Retry
            //-----------------
            MQTT_ERR_NOMEM:

              //Create Log: Unsubscribe failed, no space in message buffer

              tmpPara := to_dint(iThisMID);

              Logging_InterfLog(usLevel     :=  MQTTCLIENTINTERFACE_LOGGING_LEVEL_ERR,
                                dMsgGroup   :=  MQCLIINF_LOG_ERROR_UNSUBSCRIBE_UNSUB_FAILED_NOMEM_GRP,
                                dMsgNbr     :=  MQCLIINF_LOG_ERROR_UNSUBSCRIBE_UNSUB_FAILED_NOMEM_MSG,
                                pMsg        :=  MQCLIINF_LOG_ERROR_UNSUBSCRIBE_UNSUB_FAILED_NOMEM_TEXT,
                                pPara1      :=  #udApplMsgID$DINT,
                                pPara2      :=  #tmpPara,
                                pPara3      :=  NIL,
                                pPara4      :=  NIL);
          //All other
          else

            tmpPara := to_dint(retCode);

            Logging_InterfLog(usLevel     :=  MQTTCLIENTINTERFACE_LOGGING_LEVEL_ERR,
                              dMsgGroup   :=  MQCLIINF_LOG_ERROR_UNSUBSCRIBE_UNSUB_FAILED_GRP,
                              dMsgNbr     :=  MQCLIINF_LOG_ERROR_UNSUBSCRIBE_UNSUB_FAILED_MSG,
                              pMsg        :=  MQCLIINF_LOG_ERROR_UNSUBSCRIBE_UNSUB_FAILED_TEXT,
                              pPara1      :=  #tmpPara,
                              pPara2      :=  NIL,
                              pPara3      :=  NIL,
                              pPara4      :=  NIL);

          end_case;

          return;

        //Someone else is still subscribed to this data.
        else

          //Perform the Unsubscribed callback for this entry if it is set
          //(Even though we did not send an Unsubscribe Request we must let the requesting party know that we handled their request)
          if pPubSubEntry^.Callback.pThis   &
             pPubSubEntry^.Callback.pMethod then

            pPubSubEntry^.Callback.pMethod$PubSub_Callback(pThis        :=  pPubSubEntry^.Callback.pThis,
                                                           MsgType      :=  PSRC_Unsubscribed,
                                                           iMid         :=  pPubSubEntry^.iUnsubMid,
                                                           iGrantedQoS  :=  -1,
                                                           pMessage     :=  NIL);

          //If this is the MQTTTopic Class
          elsif pPubSubEntry^.Callback.pThis          &
                pPubSubEntry^.Callback.pMethod = NIL  then

            pPubSubEntry^.Callback.pThis$^MQTTTopic^.PubSubData(MsgType     :=  PSRC_Unsubscribed,
                                                                iMid        :=  pPubSubEntry^.iUnsubMid,
                                                                iGrantedQoS :=  -1,
                                                                pMessage    :=  NIL);

          end_if;

          //Remove this entry from the PubSubList
          if Config.pPubSubConfig^.PubSubList.udNumEntries - 1 > udCount then

            SigCLib.MemCpy( dst0  :=  pPubSubEntry,
                            src0  :=  (pPubSubEntry$UDINT + sizeof(t_s_PubSubEntry))$^void,
                            len0  :=  (sizeof(t_s_PubSubEntry) * (Config.pPubSubConfig^.PubSubList.udNumEntries - 1 - udCount)));

          end_if;

          Config.pPubSubConfig^.PubSubList.udNumEntries -= 1;

          //Return Success
          retCode := MQTTClient::MQTT_ERR_SUCCESS;
          return;

        end_if;

      end_if;

      pPubSubEntry$UDINT += sizeof(t_s_PubSubEntry);

    end_for;

    //Create Log: Failed to perform Unsubscribe command, Could not find the Subscription in the PubSubList.

    tmpPara := to_dint(pMid^);

    Logging_InterfLog(usLevel     :=  MQTTCLIENTINTERFACE_LOGGING_LEVEL_ERR,
                      dMsgGroup   :=  MQCLIINF_LOG_ERROR_UNSUBSCRIBE_UNSUB_FAILED_NOT_FOUND_GRP,
                      dMsgNbr     :=  MQCLIINF_LOG_ERROR_UNSUBSCRIBE_UNSUB_FAILED_NOT_FOUND_MSG,
                      pMsg        :=  MQCLIINF_LOG_ERROR_UNSUBSCRIBE_UNSUB_FAILED_NOT_FOUND_TEXT,
                      pPara1      :=  pApplMsgID$^DINT,
                      pPara2      :=  #tmpPara,
                      pPara3      :=  NIL,
                      pPara4      :=  NIL);

    Diagnostic_Event( Event   :=  DL_UnsubFail,
                      udValue :=  0);

  //Input values not OK
  else

    //Create Log: Failed to perform Unsubscribe Command, Input values are not OK

    Logging_InterfLog(usLevel     :=  MQTTCLIENTINTERFACE_LOGGING_LEVEL_ERR,
                      dMsgGroup   :=  MQCLIINF_LOG_ERROR_UNSUBSCRIBE_UNSUB_FAILED_INPUT_GRP,
                      dMsgNbr     :=  MQCLIINF_LOG_ERROR_UNSUBSCRIBE_UNSUB_FAILED_INPUT_MSG,
                      pMsg        :=  MQCLIINF_LOG_ERROR_UNSUBSCRIBE_UNSUB_FAILED_INPUT_TEXT,
                      pPara1      :=  NIL,
                      pPara2      :=  NIL,
                      pPara3      :=  NIL,
                      pPara4      :=  NIL);

    Diagnostic_Event( Event   :=  DL_UnsubFail,
                      udValue :=  0);

  end_if;

END_FUNCTION

FUNCTION GLOBAL MQTTClient_Interface::MQTT_SetCleanSession
	VAR_OUTPUT
		bOK 	: BOOL;
	END_VAR

  //Assume Fail
  bOK := FALSE;

  //If the state is OK
  if (InterfaceState = MCIS_Ready)              |
     (InterfaceState = MCIS_Connected)          |
     (InterfaceState = MCIS_WaitForConnection)  |
     (InterfaceState = MCIS_Reconnecting)       then

    //if the Pub Sub List is ready
    if Config.pPubSubConfig then

      Config.pPubSubConfig^.PubSubList.udNumEntries := 0;

      SigCLib.MemSet( dst :=  Config.pPubSubConfig^.PubSubList.pEntries,
                      c   :=  0x00,
                      len :=  sizeof(t_s_PubSubEntry)*Config.pPubSubConfig^.PubSubList.udMaxEntries);

    //PubSubList not Ready
    else

      //Create Log: Tried to Clean the session, Pubsub list not inititialised.

      Logging_InterfLog(usLevel     :=  MQTTCLIENTINTERFACE_LOGGING_LEVEL_ERR,
                        dMsgGroup   :=  MQCLIINF_LOG_ERROR_CLEANSESSION_PUBSUB_NOT_INITED_GRP,
                        dMsgNbr     :=  MQCLIINF_LOG_ERROR_CLEANSESSION_PUBSUB_NOT_INITED_MSG,
                        pMsg        :=  MQCLIINF_LOG_ERROR_CLEANSESSION_PUBSUB_NOT_INITED_TEXT,
                        pPara1      :=  NIL,
                        pPara2      :=  NIL,
                        pPara3      :=  NIL,
                        pPara4      :=  NIL);

    end_if;

    Config.iNextSubMID          := MQTTCLIENTINTERFACE_SUB_MID_INITVAL;
    Config.iNextPubMID          := MQTTCLIENTINTERFACE_PUB_MID_INITVAL;

    bOK := DataMap_ResetStates();

  //State not OK
  else

    //Create Log: Cannot Set clean session, the MQTT Interface is not in the correct state.

    Logging_InterfLog(usLevel     :=  MQTTCLIENTINTERFACE_LOGGING_LEVEL_ERR,
                      dMsgGroup   :=  MQCLIINF_LOG_ERROR_CLEANSESSION_FAILED_WRONG_STATE_GRP,
                      dMsgNbr     :=  MQCLIINF_LOG_ERROR_CLEANSESSION_FAILED_WRONG_STATE_MSG,
                      pMsg        :=  MQCLIINF_LOG_ERROR_CLEANSESSION_FAILED_WRONG_STATE_TEXT,
                      pPara1      :=  NIL,
                      pPara2      :=  NIL,
                      pPara3      :=  NIL,
                      pPara4      :=  NIL);

  end_if;

END_FUNCTION
//================================================================================================================================================================
//-----------------------------------------------------------------END OF INTERFACE METHODS-----------------------------------------------------------------------
//================================================================================================================================================================

//================================================================================================================================================================
//----------------------------------------------------------------------LOGGING METHODS---------------------------------------------------------------------------
//================================================================================================================================================================
FUNCTION GLOBAL MQTTClient_Interface::Logging_CreateLog
	VAR_INPUT
		usLevel 	: USINT;
		dMsgGroup 	: DINT;
		dMsgNbr 	: DINT;
		pMsg 	: ^CHAR;
		pPara1 	: ^DINT;
		pPara2 	: ^DINT;
		pPara3 	: ^DINT;
		pPara4 	: ^DINT;
		udClient 	: UDINT;(* := 0 *)
	END_VAR

  if udClient = 0 then
    return;
  end_if;

  //===================================
  //Set the Last Log Details
  //===================================
  case usLevel of

    //-----------------
    //Error
    //-----------------
    MQTT_LOG_ERR:

      DiagnosticData.LogEvents.Level_Error.dLastTopicGroup   := dMsgGroup;
      DiagnosticData.LogEvents.Level_Error.dLastTopicMessage := dMsgNbr;

      DiagnosticData.LogEvents.Level_Error.dLastGlobalGroup   := dMsgGroup;
      DiagnosticData.LogEvents.Level_Error.dLastGlobalMessage := dMsgNbr;

    //-----------------
    //Info
    //-----------------
    MQTT_LOG_INFO:

      DiagnosticData.LogEvents.Level_Info.dLastTopicGroup   := dMsgGroup;
      DiagnosticData.LogEvents.Level_Info.dLastTopicMessage := dMsgNbr;

      DiagnosticData.LogEvents.Level_Info.dLastGlobalGroup   := dMsgGroup;
      DiagnosticData.LogEvents.Level_Info.dLastGlobalMessage := dMsgNbr;

    //-----------------
    //Debug
    //-----------------
    MQTT_LOG_DEBUG:

      DiagnosticData.LogEvents.Level_Debug.dLastTopicGroup   := dMsgGroup;
      DiagnosticData.LogEvents.Level_Debug.dLastTopicMessage := dMsgNbr;

      DiagnosticData.LogEvents.Level_Debug.dLastGlobalGroup   := dMsgGroup;
      DiagnosticData.LogEvents.Level_Debug.dLastGlobalMessage := dMsgNbr;

    //-----------------
    //Warning
    //-----------------
    MQTT_LOG_WARNING:

      DiagnosticData.LogEvents.Level_Warning.dLastTopicGroup   := dMsgGroup;
      DiagnosticData.LogEvents.Level_Warning.dLastTopicMessage := dMsgNbr;

      DiagnosticData.LogEvents.Level_Warning.dLastGlobalGroup   := dMsgGroup;
      DiagnosticData.LogEvents.Level_Warning.dLastGlobalMessage := dMsgNbr;

  end_case;

  //Forward the log to the internal log function:
  Logging_InternLog(usLevel   :=  usLevel,
                    dMsgGroup :=  dMsgGroup,
                    dMsgNbr   :=  dMsgNbr,
                    pMsg      :=  pMsg,
                    pPara1    :=  pPara1,
                    pPara2    :=  pPara2,
                    pPara3    :=  pPara3,
                    pPara4    :=  pPara4);

END_FUNCTION

FUNCTION GLOBAL MQTTClient_Interface::Logging_GetLastClientEvent
	VAR_INPUT
		pGroup 	  : ^DINT;
		pMessage 	: ^DINT;
		Level 	  : DINT;
	END_VAR
	VAR_OUTPUT
		bOK 	: BOOL;
	END_VAR

  //Check if the input is OK
  bOK := pGroup & pMessage;

  if bOK then

    //================================================================
    //Based on the Event Level, write the last Event Group and Number
    //================================================================
    case level of

      //-------------
      //Error
      //-------------
      MQTTCLIENTINTERFACE_LOGGING_LEVEL_ERR:

        pGroup^   := DiagnosticData.LogEvents.Level_Error.dLastClientGroup;
        pMessage^ := DiagnosticData.LogEvents.Level_Error.dLastClientMessage;

      //-------------
      //Warning
      //-------------
      MQTTCLIENTINTERFACE_LOGGING_LEVEL_WARNING:

        pGroup^   := DiagnosticData.LogEvents.Level_Warning.dLastClientGroup;
        pMessage^ := DiagnosticData.LogEvents.Level_Warning.dLastClientMessage;

      //-------------
      //Info
      //-------------
      MQTTCLIENTINTERFACE_LOGGING_LEVEL_INFO:

        pGroup^   := DiagnosticData.LogEvents.Level_Info.dLastClientGroup;
        pMessage^ := DiagnosticData.LogEvents.Level_Info.dLastClientMessage;

      //-------------
      //Debug
      //-------------
      MQTTCLIENTINTERFACE_LOGGING_LEVEL_DEBUG:

        pGroup^   := DiagnosticData.LogEvents.Level_Debug.dLastClientGroup;
        pMessage^ := DiagnosticData.LogEvents.Level_Debug.dLastClientMessage;

    else

      bOK := FALSE;
      return;

    end_case;

  end_if;

END_FUNCTION

FUNCTION GLOBAL MQTTClient_Interface::Logging_GetLastInterfaceEvent
	VAR_INPUT
		pGroup 	  : ^DINT;
		pMessage 	: ^DINT;
		Level 	  : DINT;
	END_VAR
	VAR_OUTPUT
		bOK 	: BOOL;
	END_VAR

  //Check if the input is OK
  bOK := pGroup & pMessage;

  if bOK then

    //================================================================
    //Based on the Event Level, write the last Event Group and Number
    //================================================================
    case level of

      //-------------
      //Error
      //-------------
      MQTTCLIENTINTERFACE_LOGGING_LEVEL_ERR:

        pGroup^   := DiagnosticData.LogEvents.Level_Error.dLastInterfaceGroup;
        pMessage^ := DiagnosticData.LogEvents.Level_Error.dLastInterfaceMessage;

      //-------------
      //Warning
      //-------------
      MQTTCLIENTINTERFACE_LOGGING_LEVEL_WARNING:

        pGroup^   := DiagnosticData.LogEvents.Level_Warning.dLastInterfaceGroup;
        pMessage^ := DiagnosticData.LogEvents.Level_Warning.dLastInterfaceMessage;

      //-------------
      //Info
      //-------------
      MQTTCLIENTINTERFACE_LOGGING_LEVEL_INFO:

        pGroup^   := DiagnosticData.LogEvents.Level_Info.dLastInterfaceGroup;
        pMessage^ := DiagnosticData.LogEvents.Level_Info.dLastInterfaceMessage;

      //-------------
      //Debug
      //-------------
      MQTTCLIENTINTERFACE_LOGGING_LEVEL_DEBUG:

        pGroup^   := DiagnosticData.LogEvents.Level_Debug.dLastInterfaceGroup;
        pMessage^ := DiagnosticData.LogEvents.Level_Debug.dLastInterfaceMessage;

    else

      bOK := FALSE;
      return;

    end_case;

  end_if;

END_FUNCTION

FUNCTION GLOBAL MQTTClient_Interface::Logging_GetLastGlobalEvent
	VAR_INPUT
		pGroup 	  : ^DINT;
		pMessage 	: ^DINT;
		Level 	  : DINT;
	END_VAR
	VAR_OUTPUT
		bOK 	: BOOL;
	END_VAR

  //Check if the input is OK
  bOK := pGroup & pMessage;

  if bOK then

    //================================================================
    //Based on the Event Level, write the last Event Group and Number
    //================================================================
    case level of

      //-------------
      //Error
      //-------------
      MQTTCLIENTINTERFACE_LOGGING_LEVEL_ERR:

        pGroup^   := DiagnosticData.LogEvents.Level_Error.dLastGlobalGroup;
        pMessage^ := DiagnosticData.LogEvents.Level_Error.dLastGlobalMessage;

      //-------------
      //Warning
      //-------------
      MQTTCLIENTINTERFACE_LOGGING_LEVEL_WARNING:

        pGroup^   := DiagnosticData.LogEvents.Level_Warning.dLastGlobalGroup;
        pMessage^ := DiagnosticData.LogEvents.Level_Warning.dLastGlobalMessage;

      //-------------
      //Info
      //-------------
      MQTTCLIENTINTERFACE_LOGGING_LEVEL_INFO:

        pGroup^   := DiagnosticData.LogEvents.Level_Info.dLastGlobalGroup;
        pMessage^ := DiagnosticData.LogEvents.Level_Info.dLastGlobalMessage;

      //-------------
      //Debug
      //-------------
      MQTTCLIENTINTERFACE_LOGGING_LEVEL_DEBUG:

        pGroup^   := DiagnosticData.LogEvents.Level_Debug.dLastGlobalGroup;
        pMessage^ := DiagnosticData.LogEvents.Level_Debug.dLastGlobalMessage;

    else

      bOK := FALSE;
      return;

    end_case;

  end_if;

END_FUNCTION

FUNCTION GLOBAL MQTTClient_Interface::Logging_GetLastTopicEvent
	VAR_INPUT
		pGroup 	  : ^DINT;
		pMessage 	: ^DINT;
		Level 	  : DINT;
	END_VAR
	VAR_OUTPUT
		bOK 	: BOOL;
	END_VAR

  //Check if the input is OK
  bOK := pGroup & pMessage;

  if bOK then

    //================================================================
    //Based on the Event Level, write the last Event Group and Number
    //================================================================
    case level of

      //-------------
      //Error
      //-------------
      MQTTCLIENTINTERFACE_LOGGING_LEVEL_ERR:

        pGroup^   := DiagnosticData.LogEvents.Level_Error.dLastTopicGroup;
        pMessage^ := DiagnosticData.LogEvents.Level_Error.dLastTopicMessage;

      //-------------
      //Warning
      //-------------
      MQTTCLIENTINTERFACE_LOGGING_LEVEL_WARNING:

        pGroup^   := DiagnosticData.LogEvents.Level_Warning.dLastTopicGroup;
        pMessage^ := DiagnosticData.LogEvents.Level_Warning.dLastTopicMessage;

      //-------------
      //Info
      //-------------
      MQTTCLIENTINTERFACE_LOGGING_LEVEL_INFO:

        pGroup^   := DiagnosticData.LogEvents.Level_Info.dLastTopicGroup;
        pMessage^ := DiagnosticData.LogEvents.Level_Info.dLastTopicMessage;

      //-------------
      //Debug
      //-------------
      MQTTCLIENTINTERFACE_LOGGING_LEVEL_DEBUG:

        pGroup^   := DiagnosticData.LogEvents.Level_Debug.dLastTopicGroup;
        pMessage^ := DiagnosticData.LogEvents.Level_Debug.dLastTopicMessage;

    else

      bOK := FALSE;
      return;

    end_case;

  end_if;

END_FUNCTION

FUNCTION MQTTClient_Interface::Logging_InterfLog
	VAR_INPUT
		usLevel 	: USINT;
		dMsgGroup 	: DINT;
		dMsgNbr 	: DINT;
		pMsg 	: ^CHAR;
		pPara1 	: ^DINT;
		pPara2 	: ^DINT;
		pPara3 	: ^DINT;
		pPara4 	: ^DINT;
	END_VAR

  //===================================
  //Set the Last Log Details
  //===================================
  case usLevel of

    //-----------------
    //Error
    //-----------------
    MQTT_LOG_ERR:

      DiagnosticData.LogEvents.Level_Error.dLastInterfaceGroup  := dMsgGroup;
      DiagnosticData.LogEvents.Level_Error.dLastInterfaceMessage := dMsgNbr;

      DiagnosticData.LogEvents.Level_Error.dLastGlobalGroup   := dMsgGroup;
      DiagnosticData.LogEvents.Level_Error.dLastGlobalMessage := dMsgNbr;

    //-----------------
    //Info
    //-----------------
    MQTT_LOG_INFO:

      DiagnosticData.LogEvents.Level_Info.dLastInterfaceGroup   := dMsgGroup;
      DiagnosticData.LogEvents.Level_Info.dLastInterfaceMessage := dMsgNbr;

      DiagnosticData.LogEvents.Level_Info.dLastGlobalGroup   := dMsgGroup;
      DiagnosticData.LogEvents.Level_Info.dLastGlobalMessage := dMsgNbr;

    //-----------------
    //Debug
    //-----------------
    MQTT_LOG_DEBUG:

      DiagnosticData.LogEvents.Level_Debug.dLastInterfaceGroup   := dMsgGroup;
      DiagnosticData.LogEvents.Level_Debug.dLastInterfaceMessage := dMsgNbr;

      DiagnosticData.LogEvents.Level_Debug.dLastGlobalGroup   := dMsgGroup;
      DiagnosticData.LogEvents.Level_Debug.dLastGlobalMessage := dMsgNbr;

    //-----------------
    //Warning
    //-----------------
    MQTT_LOG_WARNING:

      DiagnosticData.LogEvents.Level_Warning.dLastInterfaceGroup   := dMsgGroup;
      DiagnosticData.LogEvents.Level_Warning.dLastInterfaceMessage := dMsgNbr;

      DiagnosticData.LogEvents.Level_Warning.dLastGlobalGroup   := dMsgGroup;
      DiagnosticData.LogEvents.Level_Warning.dLastGlobalMessage := dMsgNbr;

  end_case;

  //Forward the log to the internal log function:
  Logging_InternLog(usLevel   :=  usLevel,
                    dMsgGroup :=  dMsgGroup,
                    dMsgNbr   :=  dMsgNbr,
                    pMsg      :=  pMsg,
                    pPara1    :=  pPara1,
                    pPara2    :=  pPara2,
                    pPara3    :=  pPara3,
                    pPara4    :=  pPara4);

END_FUNCTION

FUNCTION MQTTClient_Interface::Logging_InternLog
	VAR_INPUT
		usLevel 	: USINT;
		dMsgGroup 	: DINT;
		dMsgNbr 	: DINT;
		pMsg 	: ^CHAR;
		pPara1 	: ^DINT;
		pPara2 	: ^DINT;
		pPara3 	: ^DINT;
		pPara4 	: ^DINT;
		udClient 	: UDINT;(* := 0 *)
	END_VAR

  if udClient = 0 then
    return;
  end_if;

  //Forward Log to ComLogging
  _ComLogging.AddUserEntry( Level     :=  usLevel,
                            MsgGroup  :=  dMsgGroup,
                            MsgNbr    :=  dMsgNbr,
                            pMsg      :=  pMsg,
                            pPara1    :=  pPara1,
                            pPara2    :=  pPara2,
                            pPara3    :=  pPara3,
                            pPara4    :=  pPara4);

END_FUNCTION
//================================================================================================================================================================
//------------------------------------------------------------------END OF LOGGING METHODS------------------------------------------------------------------------
//================================================================================================================================================================

//================================================================================================================================================================
//---------------------------------------------------------------------PROCESS XML METHODS------------------------------------------------------------------------
//================================================================================================================================================================
FUNCTION MQTTClient_Interface::ProcessXML
	VAR_OUTPUT
		bOK 	: BOOL;
	END_VAR
  VAR
  	pElement : ^_XML_ELEMENT;
    bFoundElement : BOOL;
    aString : ARRAY[0..MQTTCLIENT_INT_XML_FIRST_ELEMENT_MAX_LEN] of CHAR;
  END_VAR

  //Assume Error
  bOK := bFoundElement := FALSE;

  //Check the First Element
  pElement := _XMLReader.GetFirstElement();
  if pElement = NIL       |
     pElement^.Name = NIL then
    return;
  end_if;

  //Convert the String to all upper for comparison to eliminate casing constraints
    SigCLib.StrNCpy(dst0  :=  #aString[0],
                    src0  :=  pElement^.Name,
                    count :=  MQTTCLIENT_INT_XML_FIRST_ELEMENT_MAX_LEN-1);

    aString[SigCLib.StrLen(str:=pElement^.Name)] := 0x00;

    SigCLib.StrUpr(ps1:=#aString[0]);

  //If the Root Element is OK and has Children, get first Child, else stop
  if SigCLib.StrCmp(ps1:=#aString[0], ps2:=MQTTCLIENT_INT_XML_FIRST_ELEMENT_NAME) = 0 &
     pElement^.pChildren <> NIL                                                       then

    pElement := pElement^.pChildren;

  else
    //Create Log: Root Element in XML File is invalid, cannot process.

    Logging_InterfLog(usLevel     :=  MQTTCLIENTINTERFACE_LOGGING_LEVEL_ERR,
                      dMsgGroup   :=  MQCLIINF_LOG_ERROR_XML_FAILED_ROOT_WRONG_GRP,
                      dMsgNbr     :=  MQCLIINF_LOG_ERROR_XML_FAILED_ROOT_WRONG_MSG,
                      pMsg        :=  MQCLIINF_LOG_ERROR_XML_FAILED_ROOT_WRONG_TEXT,
                      pPara1      :=  NIL,
                      pPara2      :=  NIL,
                      pPara3      :=  NIL,
                      pPara4      :=  NIL);

    return;

  end_if;

  bOK := TRUE;

  //Step through all the children of the root element and process each
  while pElement <> NIL do

    //======================================================
    //Based on the XML Config section
    //======================================================
    case ProcessXML_GetElementType(pElement:=pElement) of
      //----------------------------
      //Did Not Find Element, Ignore
      //----------------------------
      X_Unknown:

      //----------------------------
      //Config Section
      //----------------------------
      X_Config:
        bOK := ProcessXML_ProcessConfig(pElement:=pElement^.pChildren);
        if bOK = FALSE then
          //Create Log, An error occurred whilst processing the Config section of the XML Document, see Log.
        end_if;

        bFoundElement := TRUE;

      //----------------------------
      //DataMap Section
      //----------------------------
      X_DataMap:
        bOK := ProcessXML_ProcessDataMap(pElement:=pElement^.pChildren);
        if bOK = FALSE then
          //Create Log, An error occurred whilst processing the DataMap section of the XML Document, see Log.
        end_if;
        bFoundElement := TRUE;

    end_case;

    //Next Element
    pElement := pElement^.pNext;

  end_while;

  bOK := bFoundElement;

END_FUNCTION

FUNCTION MQTTClient_Interface::ProcessXML_ProcessConfig
	VAR_INPUT
		pElement 	: ^_XML_ELEMENT;
	END_VAR
	VAR_OUTPUT
		bOK 	: BOOL;
	END_VAR
  VAR
  	pThisElement : ^_XML_ELEMENT;
  END_VAR

  //Assume OK
  bOK := TRUE;

  if pElement = NIL then
    return;
  end_if;

  pThisElement := pElement;

  while pThisElement do

    //==========================================================
    //Based on the type of Element, Process the section
    //==========================================================
    case ProcessXML_ProcessConfig_GetElementType(pElement:=pThisElement) of

      //-------------------------------
      //Client ID
      //-------------------------------
      t_e_XML_Config::XC_ClientID:

        //Process ClientID
        if ProcessXML_ProcessConfig_ClientID(pElement:=pThisElement) = FALSE then
          //CreateLog: Processing ClientID Section of Configuration XML File Failed.

          Logging_InterfLog(usLevel     :=  MQTTCLIENTINTERFACE_LOGGING_LEVEL_ERR,
                            dMsgGroup   :=  MQCLIINF_LOG_ERROR_XML_CONFIG_CONFIG_NOT_OK_GRP,
                            dMsgNbr     :=  MQCLIINF_LOG_ERROR_XML_CONFIG_CONFIG_NOT_OK_MSG,
                            pMsg        :=  MQCLIINF_LOG_ERROR_XML_CONFIG_CONFIG_NOT_OK_TEXT,
                            pPara1      :=  NIL,
                            pPara2      :=  NIL,
                            pPara3      :=  NIL,
                            pPara4      :=  NIL);

          bOK := FALSE;
        end_if;

      //-------------------------------
      //Connection
      //-------------------------------
      t_e_XML_Config::XC_Connection:

        if ProcessXML_ProcessConfig_Connection(pElement:=pThisElement) = FALSE then
          //CreateLog: Processing Connection Section of Configuration XML File Failed.

          Logging_InterfLog(usLevel     :=  MQTTCLIENTINTERFACE_LOGGING_LEVEL_ERR,
                            dMsgGroup   :=  MQCLIINF_LOG_ERROR_XML_CONFIG_CONNECTION_NOT_OK_GRP,
                            dMsgNbr     :=  MQCLIINF_LOG_ERROR_XML_CONFIG_CONNECTION_NOT_OK_MSG,
                            pMsg        :=  MQCLIINF_LOG_ERROR_XML_CONFIG_CONNECTION_NOT_OK_TEXT,
                            pPara1      :=  NIL,
                            pPara2      :=  NIL,
                            pPara3      :=  NIL,
                            pPara4      :=  NIL);

          bOK := FALSE;
        end_if;

      //-------------------------------
      //Will
      //-------------------------------
      t_e_XML_Config::XC_Will:

        if ProcessXML_ProcessConfig_Will(pElement:=pThisElement) = FALSE then
          //CreateLog: Processing Will Section of Configuration XML File Failed.

          Logging_InterfLog(usLevel     :=  MQTTCLIENTINTERFACE_LOGGING_LEVEL_ERR,
                            dMsgGroup   :=  MQCLIINF_LOG_ERROR_XML_CONFIG_WILL_NOT_OK_GRP,
                            dMsgNbr     :=  MQCLIINF_LOG_ERROR_XML_CONFIG_WILL_NOT_OK_MSG,
                            pMsg        :=  MQCLIINF_LOG_ERROR_XML_CONFIG_WILL_NOT_OK_TEXT,
                            pPara1      :=  NIL,
                            pPara2      :=  NIL,
                            pPara3      :=  NIL,
                            pPara4      :=  NIL);
          bOK := FALSE;
        end_if;

      //-------------------------------
      //Reconnection
      //-------------------------------
      t_e_XML_Config::XC_Reconnection:

        if ProcessXML_ProcessConfig_Reconnection(pElement:=pThisElement) = FALSE then
          //CreateLog: Processing Reonnection Section of Configuration XML File Failed.

          Logging_InterfLog(usLevel     :=  MQTTCLIENTINTERFACE_LOGGING_LEVEL_ERR,
                            dMsgGroup   :=  MQCLIINF_LOG_ERROR_XML_CONFIG_RECONNECT_NOT_OK_GRP,
                            dMsgNbr     :=  MQCLIINF_LOG_ERROR_XML_CONFIG_RECONNECT_NOT_OK_MSG,
                            pMsg        :=  MQCLIINF_LOG_ERROR_XML_CONFIG_RECONNECT_NOT_OK_TEXT,
                            pPara1      :=  NIL,
                            pPara2      :=  NIL,
                            pPara3      :=  NIL,
                            pPara4      :=  NIL);

          bOK := FALSE;

        end_if;

      //-------------------------------
      //TLS
      //-------------------------------
      t_e_XML_Config::XC_TLS:

        if ProcessXML_ProcessConfig_TLS(pElement:=pThisElement) = FALSE then
          //CreateLog: Processing TLS Section of Configuration XML File Failed.

          Logging_InterfLog(usLevel     :=  MQTTCLIENTINTERFACE_LOGGING_LEVEL_ERR,
                            dMsgGroup   :=  MQCLIINF_LOG_ERROR_XML_CONFIG_TLS_NOT_OK_GRP,
                            dMsgNbr     :=  MQCLIINF_LOG_ERROR_XML_CONFIG_TLS_NOT_OK_MSG,
                            pMsg        :=  MQCLIINF_LOG_ERROR_XML_CONFIG_TLS_NOT_OK_TEXT,
                            pPara1      :=  NIL,
                            pPara2      :=  NIL,
                            pPara3      :=  NIL,
                            pPara4      :=  NIL);

          bOK := FALSE;
        end_if;
